LIN {X 0,Y 491.423,Z 544.675,A -85,B 0,C 180,E1 -6389.515,E2 -6389.515} C_VEL
LIN {X 0,Y 491.33,Z 557.602,A -85,B 0,C 180,E1 -6389.873,E2 -6389.873} C_VEL
LIN {X 0,Y 491.207,Z 570.582,A -85,B 0,C 180,E1 -6390.411,E2 -6390.411} C_VEL
LIN {X 0,Y 490.93,Z 581.621,A -85,B 0,C 180,E1 -6391.027,E2 -6391.027} C_VEL
LIN {X 0,Y 490.598,Z 593.027,A -85,B 0,C 180,E1 -6391.848,E2 -6391.848} C_VEL
LIN {X 0,Y 490.2,Z 603.319,A -85,B 0,C 180,E1 -6392.775,E2 -6392.775} C_VEL
LIN {X 0,Y 489.929,Z 611.716,A -85,B 0,C 180,E1 -6393.702,E2 -6393.702} C_VEL
LIN {X 0,Y 489.605,Z 619.489,A -85,B 0,C 180,E1 -6394.736,E2 -6394.736} C_VEL
LIN {X 0,Y 489.353,Z 627.085,A -85,B 0,C 180,E1 -6395.978,E2 -6395.978} C_VEL
LIN {X 0,Y 489.038,Z 634.088,A -85,B 0,C 180,E1 -6397.433,E2 -6397.433} C_VEL
LIN {X 0,Y 488.829,Z 638.765,A -85,B 0,C 180,E1 -6398.684,E2 -6398.684} C_VEL
LIN {X 0,Y 488.661,Z 642.349,A -85,B 0,C 180,E1 -6399.94,E2 -6399.94} C_VEL
LIN {X 0,Y 488.576,Z 644.196,A -85,B 0,C 180,E1 -6400.779,E2 -6400.779} C_VEL
LIN {X 0,Y 488.544,Z 646.052,A -85,B 0,C 180,E1 -6401.981,E2 -6401.981} C_VEL
LIN {X 0,Y 488.468,Z 647.149,A -85,B 0,C 180,E1 -6403.31,E2 -6403.31} C_VEL
LIN {X 0,Y 488.452,Z 647.319,A -85,B 0,C 180,E1 -6404.16,E2 -6404.16} C_VEL
LIN {X 0,Y 488.511,Z 646.803,A -85,B 0,C 180,E1 -6405.443,E2 -6405.443} C_VEL
LIN {X 0,Y 488.57,Z 645.357,A -85,B 0,C 180,E1 -6406.721,E2 -6406.721} C_VEL
LIN {X 0,Y 488.722,Z 642.05,A -85,B 0,C 180,E1 -6408.36,E2 -6408.36} C_VEL
LIN {X 0,Y 488.93,Z 637.94,A -85,B 0,C 180,E1 -6409.744,E2 -6409.744} C_VEL
LIN {X 0,Y 489.167,Z 632.802,A -85,B 0,C 180,E1 -6411.051,E2 -6411.051} C_VEL
LIN {X 0,Y 489.426,Z 626.172,A -85,B 0,C 180,E1 -6412.368,E2 -6412.368} C_VEL
LIN {X 0,Y 489.828,Z 617.767,A -85,B 0,C 180,E1 -6413.688,E2 -6413.688} C_VEL
LIN {X 0,Y 490.199,Z 609.017,A -85,B 0,C 180,E1 -6414.795,E2 -6414.795} C_VEL
LIN {X 0,Y 490.541,Z 599.188,A -85,B 0,C 180,E1 -6415.798,E2 -6415.798} C_VEL
LIN {X 0,Y 490.907,Z 588.286,A -85,B 0,C 180,E1 -6416.692,E2 -6416.692} C_VEL
LIN {X 0,Y 491.228,Z 577.789,A -85,B 0,C 180,E1 -6417.376,E2 -6417.376} C_VEL
LIN {X 0,Y 491.424,Z 565.398,A -85,B 0,C 180,E1 -6417.997,E2 -6417.997} C_VEL
LIN {X 0,Y 491.551,Z 552.8,A -85,B 0,C 180,E1 -6418.445,E2 -6418.445} C_VEL
LIN {X 0,Y 491.61,Z 539.967,A -85,B 0,C 180,E1 -6418.732,E2 -6418.732} C_VEL
LIN {X 0,Y 491.994,Z 472.881,A -85,B 0,C 180,E1 -6419.731,E2 -6419.731} C_VEL
LIN {X 0,Y 488.922,Z 464.493,A -85,B 0,C 180,E1 -6420.005,E2 -6420.005} C_VEL
LIN {X 0,Y 488.757,Z 463.677,A -85,B 0,C 180,E1 -6420.17,E2 -6420.17} C_VEL
LIN {X 0,Y 488.732,Z 463.606,A -85,B 0,C 180,E1 -6423.484,E2 -6423.484} C_VEL
LIN {X 0,Y 488.685,Z 463.613,A -85,B 0,C 180,E1 -6426.355,E2 -6426.355} C_VEL
LIN {X 0,Y 488.704,Z 463.606,A -85,B 0,C 180,E1 -6429.255,E2 -6429.255} C_VEL
LIN {X 0,Y 488.711,Z 463.605,A -85,B 0,C 180,E1 -6431.601,E2 -6431.601} C_VEL
LIN {X 0,Y 488.706,Z 463.613,A -85,B 0,C 180,E1 -6434.804,E2 -6434.804} C_VEL
LIN {X 0,Y 488.696,Z 463.61,A -85,B 0,C 180,E1 -6437.475,E2 -6437.475} C_VEL
LIN {X 0,Y 488.738,Z 463.606,A -85,B 0,C 180,E1 -6439.677,E2 -6439.677} C_VEL
LIN {X 0,Y 488.775,Z 463.798,A -85,B 0,C 180,E1 -6442.058,E2 -6442.058} C_VEL
LIN {X 0,Y 490.787,Z 474.144,A -85,B 0,C 180,E1 -6443.831,E2 -6443.831} C_VEL
LIN {X 0,Y 490.488,Z 489.742,A -85,B 0,C 180,E1 -6446.311,E2 -6446.311} C_VEL
LIN {X 0,Y 489.94,Z 509.149,A -85,B 0,C 180,E1 -6449.394,E2 -6449.394} C_VEL
LIN {X 0,Y 489.799,Z 518.237,A -85,B 0,C 180,E1 -6450.801,E2 -6450.801} C_VEL
LIN {X 0,Y 491.769,Z 530.283,A -85,B 0,C 180,E1 -6451.078,E2 -6451.078} C_VEL
LIN {X 0,Y 491.009,Z 626.779,A -85,B 0,C 180,E1 -6452.579,E2 -6452.579} C_VEL
LIN {X 0,Y 490.736,Z 640.314,A -85,B 0,C 180,E1 -6452.955,E2 -6452.955} C_VEL
LIN {X 0,Y 490.385,Z 653.402,A -85,B 0,C 180,E1 -6453.509,E2 -6453.509} C_VEL
LIN {X 0,Y 490.075,Z 665.153,A -85,B 0,C 180,E1 -6454.177,E2 -6454.177} C_VEL
LIN {X 0,Y 489.69,Z 676.455,A -85,B 0,C 180,E1 -6455.007,E2 -6455.007} C_VEL
LIN {X 0,Y 489.259,Z 686.707,A -85,B 0,C 180,E1 -6455.947,E2 -6455.947} C_VEL
LIN {X 0,Y 488.963,Z 695.329,A -85,B 0,C 180,E1 -6456.912,E2 -6456.912} C_VEL
LIN {X 0,Y 488.674,Z 703.624,A -85,B 0,C 180,E1 -6458.042,E2 -6458.042} C_VEL
LIN {X 0,Y 488.354,Z 711.06,A -85,B 0,C 180,E1 -6459.3,E2 -6459.3} C_VEL
LIN {X 0,Y 488.216,Z 717.473,A -85,B 0,C 180,E1 -6460.665,E2 -6460.665} C_VEL
LIN {X 0,Y 488.079,Z 721.901,A -85,B 0,C 180,E1 -6461.873,E2 -6461.873} C_VEL
LIN {X 0,Y 487.931,Z 725.713,A -85,B 0,C 180,E1 -6463.258,E2 -6463.258} C_VEL
LIN {X 0,Y 487.881,Z 728.525,A -85,B 0,C 180,E1 -6464.832,E2 -6464.832} C_VEL
LIN {X 0,Y 487.862,Z 729.56,A -85,B 0,C 180,E1 -6465.825,E2 -6465.825} C_VEL
LIN {X 0,Y 487.853,Z 729.953,A -85,B 0,C 180,E1 -6466.674,E2 -6466.674} C_VEL
LIN {X 0,Y 487.866,Z 729.946,A -85,B 0,C 180,E1 -6467.521,E2 -6467.521} C_VEL
LIN {X 0,Y 487.954,Z 729.524,A -85,B 0,C 180,E1 -6468.367,E2 -6468.367} C_VEL
LIN {X 0,Y 487.944,Z 728.654,A -85,B 0,C 180,E1 -6469.208,E2 -6469.208} C_VEL
LIN {X 0,Y 487.925,Z 727.388,A -85,B 0,C 180,E1 -6470.047,E2 -6470.047} C_VEL
LIN {X 0,Y 488.016,Z 724.667,A -85,B 0,C 180,E1 -6471.303,E2 -6471.303} C_VEL
LIN {X 0,Y 488.143,Z 720.913,A -85,B 0,C 180,E1 -6472.555,E2 -6472.555} C_VEL
LIN {X 0,Y 488.281,Z 715.569,A -85,B 0,C 180,E1 -6473.911,E2 -6473.911} C_VEL
LIN {X 0,Y 488.438,Z 708.705,A -85,B 0,C 180,E1 -6475.255,E2 -6475.255} C_VEL
LIN {X 0,Y 488.753,Z 700.753,A -85,B 0,C 180,E1 -6476.497,E2 -6476.497} C_VEL
LIN {X 0,Y 489.085,Z 692.626,A -85,B 0,C 180,E1 -6477.53,E2 -6477.53} C_VEL
LIN {X 0,Y 489.444,Z 682.634,A -85,B 0,C 180,E1 -6478.56,E2 -6478.56} C_VEL
LIN {X 0,Y 489.851,Z 671.472,A -85,B 0,C 180,E1 -6479.487,E2 -6479.487} C_VEL
LIN {X 0,Y 490.217,Z 660.49,A -85,B 0,C 180,E1 -6480.206,E2 -6480.206} C_VEL
LIN {X 0,Y 490.542,Z 648.224,A -85,B 0,C 180,E1 -6480.821,E2 -6480.821} C_VEL
LIN {X 0,Y 490.786,Z 635.579,A -85,B 0,C 180,E1 -6481.282,E2 -6481.282} C_VEL
LIN {X 0,Y 490.993,Z 621.991,A -85,B 0,C 180,E1 -6481.589,E2 -6481.589} C_VEL
LIN {X 0,Y 491.668,Z 529.585,A -85,B 0,C 180,E1 -6483.035,E2 -6483.035} C_VEL
LIN {X 0,Y 489.964,Z 519.063,A -85,B 0,C 180,E1 -6483.289,E2 -6483.289} C_VEL
LIN {X 0,Y 490.304,Z 499.165,A -85,B 0,C 180,E1 -6486.378,E2 -6486.378} C_VEL
LIN {X 0,Y 490.632,Z 482.876,A -85,B 0,C 180,E1 -6488.888,E2 -6488.888} C_VEL
LIN {X 0,Y 490.643,Z 473.536,A -85,B 0,C 180,E1 -6490.315,E2 -6490.315} C_VEL
LIN {X 0,Y 488.833,Z 463.701,A -85,B 0,C 180,E1 -6491.932,E2 -6491.932} C_VEL
LIN {X 0,Y 488.784,Z 463.602,A -85,B 0,C 180,E1 -6495.554,E2 -6495.554} C_VEL
LIN {X 0,Y 488.754,Z 463.604,A -85,B 0,C 180,E1 -6498.442,E2 -6498.442} C_VEL
LIN {X 0,Y 488.715,Z 463.612,A -85,B 0,C 180,E1 -6501.071,E2 -6501.071} C_VEL
LIN {X 0,Y 488.679,Z 463.611,A -85,B 0,C 180,E1 -6503.746,E2 -6503.746} C_VEL
LIN {X 0,Y 488.756,Z 463.606,A -85,B 0,C 180,E1 -6506.933,E2 -6506.933} C_VEL
LIN {X 0,Y 488.731,Z 463.606,A -85,B 0,C 180,E1 -6509.27,E2 -6509.27} C_VEL
LIN {X 0,Y 488.711,Z 463.607,A -85,B 0,C 180,E1 -6512.147,E2 -6512.147} C_VEL
LIN {X 0,Y 488.726,Z 463.606,A -85,B 0,C 180,E1 -6515.115,E2 -6515.115} C_VEL
LIN {X 0,Y 488.688,Z 463.612,A -85,B 0,C 180,E1 -6518.2,E2 -6518.2} C_VEL
LIN {X 0,Y 488.727,Z 463.608,A -85,B 0,C 180,E1 -6520.344,E2 -6520.344} C_VEL
LIN {X 0,Y 488.692,Z 463.609,A -85,B 0,C 180,E1 -6523.654,E2 -6523.654} C_VEL
LIN {X 0,Y 488.692,Z 463.613,A -85,B 0,C 180,E1 -6526.345,E2 -6526.345} C_VEL
LIN {X 0,Y 488.741,Z 463.604,A -85,B 0,C 180,E1 -6529.676,E2 -6529.676} C_VEL
LIN {X 0,Y 488.677,Z 463.61,A -85,B 0,C 180,E1 -6532.84,E2 -6532.84} C_VEL
LIN {X 0,Y 488.725,Z 463.599,A -85,B 0,C 180,E1 -6535.885,E2 -6535.885} C_VEL
LIN {X 0,Y 488.698,Z 463.611,A -85,B 0,C 180,E1 -6538.819,E2 -6538.819} C_VEL
LIN {X 0,Y 488.799,Z 463.817,A -85,B 0,C 180,E1 -6540.334,E2 -6540.334} C_VEL
LIN {X 0,Y 492.029,Z 478.714,A -85,B 0,C 180,E1 -6542.534,E2 -6542.534} C_VEL
LIN {X 0,Y 491.86,Z 487.643,A -85,B 0,C 180,E1 -6543.707,E2 -6543.707} C_VEL
LIN {X 0,Y 491.059,Z 510.131,A -85,B 0,C 180,E1 -6546.598,E2 -6546.598} C_VEL
LIN {X 0,Y 490.338,Z 532.663,A -85,B 0,C 180,E1 -6549.441,E2 -6549.441} C_VEL
LIN {X 0,Y 489.667,Z 556.938,A -85,B 0,C 180,E1 -6552.457,E2 -6552.457} C_VEL
LIN {X 0,Y 489.448,Z 567.191,A -85,B 0,C 180,E1 -6553.696,E2 -6553.696} C_VEL
LIN {X 0,Y 491.565,Z 587.846,A -85,B 0,C 180,E1 -6554.086,E2 -6554.086} C_VEL
LIN {X 0,Y 491.001,Z 678.547,A -85,B 0,C 180,E1 -6555.439,E2 -6555.439} C_VEL
LIN {X 0,Y 490.587,Z 692.383,A -85,B 0,C 180,E1 -6555.824,E2 -6555.824} C_VEL
LIN {X 0,Y 490.217,Z 705.371,A -85,B 0,C 180,E1 -6556.368,E2 -6556.368} C_VEL
LIN {X 0,Y 489.788,Z 717.734,A -85,B 0,C 180,E1 -6557.074,E2 -6557.074} C_VEL
LIN {X 0,Y 489.444,Z 728.753,A -85,B 0,C 180,E1 -6557.876,E2 -6557.876} C_VEL
LIN {X 0,Y 488.951,Z 739.13,A -85,B 0,C 180,E1 -6558.81,E2 -6558.81} C_VEL
LIN {X 0,Y 488.72,Z 748.521,A -85,B 0,C 180,E1 -6559.853,E2 -6559.853} C_VEL
LIN {X 0,Y 488.44,Z 757.666,A -85,B 0,C 180,E1 -6561.101,E2 -6561.101} C_VEL
LIN {X 0,Y 488.243,Z 765.039,A -85,B 0,C 180,E1 -6562.347,E2 -6562.347} C_VEL
LIN {X 0,Y 488.133,Z 771.508,A -85,B 0,C 180,E1 -6563.686,E2 -6563.686} C_VEL
LIN {X 0,Y 488.082,Z 776.557,A -85,B 0,C 180,E1 -6565.042,E2 -6565.042} C_VEL
LIN {X 0,Y 488.135,Z 778.96,A -85,B 0,C 180,E1 -6565.87,E2 -6565.87} C_VEL
LIN {X 0,Y 488.074,Z 780.886,A -85,B 0,C 180,E1 -6566.697,E2 -6566.697} C_VEL
LIN {X 0,Y 488.067,Z 782.375,A -85,B 0,C 180,E1 -6567.523,E2 -6567.523} C_VEL
LIN {X 0,Y 488.009,Z 783.436,A -85,B 0,C 180,E1 -6568.348,E2 -6568.348} C_VEL
LIN {X 0,Y 487.983,Z 784.079,A -85,B 0,C 180,E1 -6569.173,E2 -6569.173} C_VEL
LIN {X 0,Y 488.043,Z 784.312,A -85,B 0,C 180,E1 -6569.999,E2 -6569.999} C_VEL
LIN {X 0,Y 487.98,Z 784.11,A -85,B 0,C 180,E1 -6570.824,E2 -6570.824} C_VEL
LIN {X 0,Y 488.003,Z 783.495,A -85,B 0,C 180,E1 -6571.649,E2 -6571.649} C_VEL
LIN {X 0,Y 488.061,Z 782.466,A -85,B 0,C 180,E1 -6572.475,E2 -6572.475} C_VEL
LIN {X 0,Y 488.067,Z 781.001,A -85,B 0,C 180,E1 -6573.301,E2 -6573.301} C_VEL
LIN {X 0,Y 488.05,Z 777.918,A -85,B 0,C 180,E1 -6574.541,E2 -6574.541} C_VEL
LIN {X 0,Y 488.18,Z 772.758,A -85,B 0,C 180,E1 -6576.046,E2 -6576.046} C_VEL
LIN {X 0,Y 488.205,Z 766.364,A -85,B 0,C 180,E1 -6577.443,E2 -6577.443} C_VEL
LIN {X 0,Y 488.389,Z 759.172,A -85,B 0,C 180,E1 -6578.689,E2 -6578.689} C_VEL
LIN {X 0,Y 488.632,Z 750.351,A -85,B 0,C 180,E1 -6579.937,E2 -6579.937} C_VEL
LIN {X 0,Y 488.956,Z 741.346,A -85,B 0,C 180,E1 -6580.977,E2 -6580.977} C_VEL
LIN {X 0,Y 489.354,Z 731.482,A -85,B 0,C 180,E1 -6581.913,E2 -6581.913} C_VEL
LIN {X 0,Y 489.709,Z 720.852,A -85,B 0,C 180,E1 -6582.735,E2 -6582.735} C_VEL
LIN {X 0,Y 490.113,Z 708.68,A -85,B 0,C 180,E1 -6583.473,E2 -6583.473} C_VEL
LIN {X 0,Y 490.512,Z 696.213,A -85,B 0,C 180,E1 -6584.043,E2 -6584.043} C_VEL
LIN {X 0,Y 490.892,Z 683.439,A -85,B 0,C 180,E1 -6584.455,E2 -6584.455} C_VEL
LIN {X 0,Y 491.073,Z 670.047,A -85,B 0,C 180,E1 -6584.715,E2 -6584.715} C_VEL
LIN {X 0,Y 491.533,Z 585.726,A -85,B 0,C 180,E1 -6585.951,E2 -6585.951} C_VEL
LIN {X 0,Y 489.464,Z 567.613,A -85,B 0,C 180,E1 -6586.301,E2 -6586.301} C_VEL
LIN {X 0,Y 489.986,Z 545.924,A -85,B 0,C 180,E1 -6588.965,E2 -6588.965} C_VEL
LIN {X 0,Y 490.885,Z 517.599,A -85,B 0,C 180,E1 -6592.517,E2 -6592.517} C_VEL
LIN {X 0,Y 491.631,Z 493.909,A -85,B 0,C 180,E1 -6595.531,E2 -6595.531} C_VEL
LIN {X 0,Y 492.066,Z 478.853,A -85,B 0,C 180,E1 -6597.477,E2 -6597.477} C_VEL
LIN {X 0,Y 488.75,Z 463.732,A -85,B 0,C 180,E1 -6599.666,E2 -6599.666} C_VEL
LIN {X 0,Y 488.73,Z 463.606,A -85,B 0,C 180,E1 -6603.121,E2 -6603.121} C_VEL
LIN {X 0,Y 488.658,Z 463.619,A -85,B 0,C 180,E1 -6606.132,E2 -6606.132} C_VEL
LIN {X 0,Y 488.68,Z 463.608,A -85,B 0,C 180,E1 -6609.254,E2 -6609.254} C_VEL
LIN {X 0,Y 488.658,Z 463.615,A -85,B 0,C 180,E1 -6612.527,E2 -6612.527} C_VEL
LIN {X 0,Y 488.692,Z 463.606,A -85,B 0,C 180,E1 -6615.196,E2 -6615.196} C_VEL
LIN {X 0,Y 488.67,Z 463.613,A -85,B 0,C 180,E1 -6618.58,E2 -6618.58} C_VEL
LIN {X 0,Y 488.664,Z 463.612,A -85,B 0,C 180,E1 -6621.798,E2 -6621.798} C_VEL
LIN {X 0,Y 488.711,Z 463.604,A -85,B 0,C 180,E1 -6625.051,E2 -6625.051} C_VEL
LIN {X 0,Y 488.692,Z 463.611,A -85,B 0,C 180,E1 -6628.045,E2 -6628.045} C_VEL
LIN {X 0,Y 488.71,Z 463.607,A -85,B 0,C 180,E1 -6630.728,E2 -6630.728} C_VEL
LIN {X 0,Y 488.723,Z 463.603,A -85,B 0,C 180,E1 -6633.526,E2 -6633.526} C_VEL
LIN {X 0,Y 488.659,Z 463.617,A -85,B 0,C 180,E1 -6636.252,E2 -6636.252} C_VEL
LIN {X 0,Y 488.733,Z 463.601,A -85,B 0,C 180,E1 -6639.175,E2 -6639.175} C_VEL
LIN {X 0,Y 488.714,Z 463.613,A -85,B 0,C 180,E1 -6642.422,E2 -6642.422} C_VEL
LIN {X 0,Y 488.747,Z 463.601,A -85,B 0,C 180,E1 -6644.999,E2 -6644.999} C_VEL
LIN {X 0,Y 488.795,Z 463.601,A -85,B 0,C 180,E1 -6648.387,E2 -6648.387} C_VEL
LIN {X 0,Y 488.802,Z 463.593,A -85,B 0,C 180,E1 -6651.733,E2 -6651.733} C_VEL
LIN {X 0,Y 488.829,Z 463.594,A -85,B 0,C 180,E1 -6654.224,E2 -6654.224} C_VEL
LIN {X 0,Y 488.945,Z 463.575,A -85,B 0,C 180,E1 -6657.528,E2 -6657.528} C_VEL
LIN {X 0,Y 488.962,Z 463.577,A -85,B 0,C 180,E1 -6660.823,E2 -6660.823} C_VEL
LIN {X 0,Y 488.946,Z 463.582,A -85,B 0,C 180,E1 -6662.471,E2 -6662.471} C_VEL
LIN {X 0,Y 488.833,Z 463.589,A -85,B 0,C 180,E1 -6665.776,E2 -6665.776} C_VEL
LIN {X 0,Y 488.804,Z 463.596,A -85,B 0,C 180,E1 -6668.266,E2 -6668.266} C_VEL
LIN {X 0,Y 488.794,Z 463.593,A -85,B 0,C 180,E1 -6671.612,E2 -6671.612} C_VEL
LIN {X 0,Y 488.75,Z 463.603,A -85,B 0,C 180,E1 -6675,E2 -6675} C_VEL
LIN {X 0,Y 488.74,Z 463.605,A -85,B 0,C 180,E1 -6678.442,E2 -6678.442} C_VEL
LIN {X 0,Y 488.694,Z 463.61,A -85,B 0,C 180,E1 -6681.071,E2 -6681.071} C_VEL
LIN {X 0,Y 488.679,Z 463.608,A -85,B 0,C 180,E1 -6683.746,E2 -6683.746} C_VEL
LIN {X 0,Y 488.785,Z 463.601,A -85,B 0,C 180,E1 -6686.946,E2 -6686.946} C_VEL
LIN {X 0,Y 488.696,Z 463.609,A -85,B 0,C 180,E1 -6690.364,E2 -6690.364} C_VEL
LIN {X 0,Y 488.723,Z 463.603,A -85,B 0,C 180,E1 -6693.485,E2 -6693.485} C_VEL
LIN {X 0,Y 488.676,Z 463.611,A -85,B 0,C 180,E1 -6696.356,E2 -6696.356} C_VEL
LIN {X 0,Y 488.689,Z 463.61,A -85,B 0,C 180,E1 -6699.255,E2 -6699.255} C_VEL
LIN {X 0,Y 488.711,Z 463.604,A -85,B 0,C 180,E1 -6701.603,E2 -6701.603} C_VEL
LIN {X 0,Y 488.7,Z 463.613,A -85,B 0,C 180,E1 -6704.802,E2 -6704.802} C_VEL
LIN {X 0,Y 488.723,Z 463.604,A -85,B 0,C 180,E1 -6707.48,E2 -6707.48} C_VEL
LIN {X 0,Y 488.739,Z 463.607,A -85,B 0,C 180,E1 -6710.752,E2 -6710.752} C_VEL
LIN {X 0,Y 488.674,Z 463.608,A -85,B 0,C 180,E1 -6713.87,E2 -6713.87} C_VEL
LIN {X 0,Y 488.731,Z 463.609,A -85,B 0,C 180,E1 -6716.879,E2 -6716.879} C_VEL
LIN {X 0,Y 488.716,Z 463.603,A -85,B 0,C 180,E1 -6719.782,E2 -6719.782} C_VEL
LIN {X 0,Y 488.785,Z 463.603,A -85,B 0,C 180,E1 -6723.058,E2 -6723.058} C_VEL
LIN {X 0,Y 488.736,Z 463.602,A -85,B 0,C 180,E1 -6724.363,E2 -6724.363} C_VEL
LIN {X 0,Y 488.093,Z 463.69,A -85,B 0,C 180,E1 -6725.051,E2 -6725.051} C_VEL
LIN {X 0,Y 485.223,Z 464.043,A -85,B 0,C 180,E1 -6726.168,E2 -6726.168} C_VEL
LIN {X 0,Y 482.776,Z 464.352,A -85,B 0,C 180,E1 -6727.068,E2 -6727.068} C_VEL
LIN {X 0,Y 481.718,Z 464.476,A -85,B 0,C 180,E1 -6727.763,E2 -6727.763} C_VEL
LIN {X 0,Y 481.63,Z 464.486,A -85,B 0,C 180,E1 -6727.999,E2 -6727.999} C_VEL
LIN {X 0,Y 481.702,Z 464.478,A -85,B 0,C 180,E1 -6730.395,E2 -6730.395} C_VEL
LIN {X 0,Y 481.687,Z 464.487,A -85,B 0,C 180,E1 -6733.035,E2 -6733.035} C_VEL
LIN {X 0,Y 481.686,Z 464.481,A -85,B 0,C 180,E1 -6735.64,E2 -6735.64} C_VEL
LIN {X 0,Y 481.747,Z 464.471,A -85,B 0,C 180,E1 -6738.217,E2 -6738.217} C_VEL
LIN {X 0,Y 481.76,Z 464.475,A -85,B 0,C 180,E1 -6741.613,E2 -6741.613} C_VEL
LIN {X 0,Y 481.817,Z 464.467,A -85,B 0,C 180,E1 -6744.141,E2 -6744.141} C_VEL
LIN {X 0,Y 481.885,Z 464.583,A -85,B 0,C 180,E1 -6747.839,E2 -6747.839} C_VEL
LIN {X 0,Y 482.07,Z 465.64,A -85,B 0,C 180,E1 -6747.996,E2 -6747.996} C_VEL
LIN {X 0,Y 484.988,Z 474.293,A -85,B 0,C 180,E1 -6748.235,E2 -6748.235} C_VEL
LIN {X 0,Y 484.58,Z 545.83,A -85,B 0,C 180,E1 -6749.326,E2 -6749.326} C_VEL
LIN {X 0,Y 484.488,Z 558.693,A -85,B 0,C 180,E1 -6749.69,E2 -6749.69} C_VEL
LIN {X 0,Y 484.358,Z 571.103,A -85,B 0,C 180,E1 -6750.209,E2 -6750.209} C_VEL
LIN {X 0,Y 484.066,Z 582.267,A -85,B 0,C 180,E1 -6750.833,E2 -6750.833} C_VEL
LIN {X 0,Y 483.712,Z 593.755,A -85,B 0,C 180,E1 -6751.667,E2 -6751.667} C_VEL
LIN {X 0,Y 483.302,Z 604.094,A -85,B 0,C 180,E1 -6752.606,E2 -6752.606} C_VEL
LIN {X 0,Y 483.018,Z 612.523,A -85,B 0,C 180,E1 -6753.547,E2 -6753.547} C_VEL
LIN {X 0,Y 482.672,Z 620.324,A -85,B 0,C 180,E1 -6754.595,E2 -6754.595} C_VEL
LIN {X 0,Y 482.376,Z 627.962,A -85,B 0,C 180,E1 -6755.855,E2 -6755.855} C_VEL
LIN {X 0,Y 482.083,Z 634.595,A -85,B 0,C 180,E1 -6757.239,E2 -6757.239} C_VEL
LIN {X 0,Y 481.806,Z 640.371,A -85,B 0,C 180,E1 -6758.812,E2 -6758.812} C_VEL
LIN {X 0,Y 481.634,Z 643.8,A -85,B 0,C 180,E1 -6760.086,E2 -6760.086} C_VEL
LIN {X 0,Y 481.538,Z 645.51,A -85,B 0,C 180,E1 -6760.939,E2 -6760.939} C_VEL
LIN {X 0,Y 481.522,Z 647.165,A -85,B 0,C 180,E1 -6762.072,E2 -6762.072} C_VEL
LIN {X 0,Y 481.455,Z 648.2,A -85,B 0,C 180,E1 -6763.508,E2 -6763.508} C_VEL
LIN {X 0,Y 481.426,Z 648.271,A -85,B 0,C 180,E1 -6764.371,E2 -6764.371} C_VEL
LIN {X 0,Y 481.496,Z 647.711,A -85,B 0,C 180,E1 -6765.562,E2 -6765.562} C_VEL
LIN {X 0,Y 481.58,Z 646.015,A -85,B 0,C 180,E1 -6766.971,E2 -6766.971} C_VEL
LIN {X 0,Y 481.738,Z 642.857,A -85,B 0,C 180,E1 -6768.51,E2 -6768.51} C_VEL
LIN {X 0,Y 481.99,Z 638.244,A -85,B 0,C 180,E1 -6770.04,E2 -6770.04} C_VEL
LIN {X 0,Y 482.244,Z 632.868,A -85,B 0,C 180,E1 -6771.368,E2 -6771.368} C_VEL
LIN {X 0,Y 482.591,Z 626.011,A -85,B 0,C 180,E1 -6772.702,E2 -6772.702} C_VEL
LIN {X 0,Y 482.943,Z 618.522,A -85,B 0,C 180,E1 -6773.876,E2 -6773.876} C_VEL
LIN {X 0,Y 483.322,Z 610.208,A -85,B 0,C 180,E1 -6774.943,E2 -6774.943} C_VEL
LIN {X 0,Y 483.687,Z 600.444,A -85,B 0,C 180,E1 -6775.96,E2 -6775.96} C_VEL
LIN {X 0,Y 484.085,Z 589.615,A -85,B 0,C 180,E1 -6776.865,E2 -6776.865} C_VEL
LIN {X 0,Y 484.411,Z 579.41,A -85,B 0,C 180,E1 -6777.547,E2 -6777.547} C_VEL
LIN {X 0,Y 484.645,Z 568.151,A -85,B 0,C 180,E1 -6778.137,E2 -6778.137} C_VEL
LIN {X 0,Y 484.766,Z 555.689,A -85,B 0,C 180,E1 -6778.613,E2 -6778.613} C_VEL
LIN {X 0,Y 484.823,Z 542.482,A -85,B 0,C 180,E1 -6778.934,E2 -6778.934} C_VEL
LIN {X 0,Y 485.23,Z 474.35,A -85,B 0,C 180,E1 -6779.969,E2 -6779.969} C_VEL
LIN {X 0,Y 481.901,Z 465.577,A -85,B 0,C 180,E1 -6780.255,E2 -6780.255} C_VEL
LIN {X 0,Y 481.681,Z 464.581,A -85,B 0,C 180,E1 -6780.424,E2 -6780.424} C_VEL
LIN {X 0,Y 481.678,Z 464.484,A -85,B 0,C 180,E1 -6783.73,E2 -6783.73} C_VEL
LIN {X 0,Y 481.629,Z 464.492,A -85,B 0,C 180,E1 -6786.748,E2 -6786.748} C_VEL
LIN {X 0,Y 481.681,Z 464.479,A -85,B 0,C 180,E1 -6789.941,E2 -6789.941} C_VEL
LIN {X 0,Y 481.636,Z 464.491,A -85,B 0,C 180,E1 -6793.148,E2 -6793.148} C_VEL
LIN {X 0,Y 481.658,Z 464.485,A -85,B 0,C 180,E1 -6795.642,E2 -6795.642} C_VEL
LIN {X 0,Y 481.661,Z 464.491,A -85,B 0,C 180,E1 -6798.959,E2 -6798.959} C_VEL
LIN {X 0,Y 481.738,Z 464.702,A -85,B 0,C 180,E1 -6801.864,E2 -6801.864} C_VEL
LIN {X 0,Y 483.873,Z 475.473,A -85,B 0,C 180,E1 -6803.711,E2 -6803.711} C_VEL
LIN {X 0,Y 483.569,Z 491.007,A -85,B 0,C 180,E1 -6806.203,E2 -6806.203} C_VEL
LIN {X 0,Y 483.022,Z 509.39,A -85,B 0,C 180,E1 -6809.145,E2 -6809.145} C_VEL
LIN {X 0,Y 482.83,Z 518.311,A -85,B 0,C 180,E1 -6810.546,E2 -6810.546} C_VEL
LIN {X 0,Y 484.098,Z 525.738,A -85,B 0,C 180,E1 -6810.743,E2 -6810.743} C_VEL
LIN {X 0,Y 484.911,Z 531.562,A -85,B 0,C 180,E1 -6810.865,E2 -6810.865} C_VEL
LIN {X 0,Y 484.112,Z 626.805,A -85,B 0,C 180,E1 -6812.378,E2 -6812.378} C_VEL
LIN {X 0,Y 483.834,Z 639.961,A -85,B 0,C 180,E1 -6812.741,E2 -6812.741} C_VEL
LIN {X 0,Y 483.48,Z 652.693,A -85,B 0,C 180,E1 -6813.275,E2 -6813.275} C_VEL
LIN {X 0,Y 483.139,Z 665.57,A -85,B 0,C 180,E1 -6814.01,E2 -6814.01} C_VEL
LIN {X 0,Y 482.72,Z 677.046,A -85,B 0,C 180,E1 -6814.868,E2 -6814.868} C_VEL
LIN {X 0,Y 482.271,Z 687.112,A -85,B 0,C 180,E1 -6815.804,E2 -6815.804} C_VEL
LIN {X 0,Y 481.955,Z 695.982,A -85,B 0,C 180,E1 -6816.814,E2 -6816.814} C_VEL
LIN {X 0,Y 481.655,Z 704.031,A -85,B 0,C 180,E1 -6817.931,E2 -6817.931} C_VEL
LIN {X 0,Y 481.342,Z 711.135,A -85,B 0,C 180,E1 -6819.143,E2 -6819.143} C_VEL
LIN {X 0,Y 481.171,Z 716.953,A -85,B 0,C 180,E1 -6820.371,E2 -6820.371} C_VEL
LIN {X 0,Y 481.017,Z 722.101,A -85,B 0,C 180,E1 -6821.752,E2 -6821.752} C_VEL
LIN {X 0,Y 480.875,Z 725.61,A -85,B 0,C 180,E1 -6823.005,E2 -6823.005} C_VEL
LIN {X 0,Y 480.83,Z 727.465,A -85,B 0,C 180,E1 -6823.877,E2 -6823.877} C_VEL
LIN {X 0,Y 480.796,Z 728.836,A -85,B 0,C 180,E1 -6824.745,E2 -6824.745} C_VEL
LIN {X 0,Y 480.795,Z 729.792,A -85,B 0,C 180,E1 -6825.612,E2 -6825.612} C_VEL
LIN {X 0,Y 480.76,Z 730.306,A -85,B 0,C 180,E1 -6826.474,E2 -6826.474} C_VEL
LIN {X 0,Y 480.779,Z 730.374,A -85,B 0,C 180,E1 -6827.334,E2 -6827.334} C_VEL
LIN {X 0,Y 480.859,Z 729.977,A -85,B 0,C 180,E1 -6828.309,E2 -6828.309} C_VEL
LIN {X 0,Y 480.859,Z 728.102,A -85,B 0,C 180,E1 -6829.899,E2 -6829.899} C_VEL
LIN {X 0,Y 480.941,Z 725.524,A -85,B 0,C 180,E1 -6831.174,E2 -6831.174} C_VEL
LIN {X 0,Y 481.067,Z 721.918,A -85,B 0,C 180,E1 -6832.445,E2 -6832.445} C_VEL
LIN {X 0,Y 481.224,Z 716.591,A -85,B 0,C 180,E1 -6833.856,E2 -6833.856} C_VEL
LIN {X 0,Y 481.383,Z 710.119,A -85,B 0,C 180,E1 -6835.185,E2 -6835.185} C_VEL
LIN {X 0,Y 481.681,Z 702.374,A -85,B 0,C 180,E1 -6836.445,E2 -6836.445} C_VEL
LIN {X 0,Y 482.039,Z 694.484,A -85,B 0,C 180,E1 -6837.493,E2 -6837.493} C_VEL
LIN {X 0,Y 482.397,Z 684.909,A -85,B 0,C 180,E1 -6838.539,E2 -6838.539} C_VEL
LIN {X 0,Y 482.808,Z 674.153,A -85,B 0,C 180,E1 -6839.479,E2 -6839.479} C_VEL
LIN {X 0,Y 483.255,Z 662.086,A -85,B 0,C 180,E1 -6840.313,E2 -6840.313} C_VEL
LIN {X 0,Y 483.63,Z 650.191,A -85,B 0,C 180,E1 -6840.937,E2 -6840.937} C_VEL
LIN {X 0,Y 483.907,Z 636.515,A -85,B 0,C 180,E1 -6841.457,E2 -6841.457} C_VEL
LIN {X 0,Y 484.092,Z 623.457,A -85,B 0,C 180,E1 -6841.768,E2 -6841.768} C_VEL
LIN {X 0,Y 484.876,Z 530.321,A -85,B 0,C 180,E1 -6843.259,E2 -6843.259} C_VEL
LIN {X 0,Y 483.077,Z 519.738,A -85,B 0,C 180,E1 -6843.519,E2 -6843.519} C_VEL
LIN {X 0,Y 483.07,Z 516.568,A -85,B 0,C 180,E1 -6843.963,E2 -6843.963} C_VEL
LIN {X 0,Y 483.58,Z 495.339,A -85,B 0,C 180,E1 -6847.306,E2 -6847.306} C_VEL
LIN {X 0,Y 483.894,Z 476.198,A -85,B 0,C 180,E1 -6850.249,E2 -6850.249} C_VEL
LIN {X 0,Y 481.801,Z 464.684,A -85,B 0,C 180,E1 -6852.123,E2 -6852.123} C_VEL
LIN {X 0,Y 481.732,Z 464.48,A -85,B 0,C 180,E1 -6855.658,E2 -6855.658} C_VEL
LIN {X 0,Y 481.715,Z 464.483,A -85,B 0,C 180,E1 -6858.722,E2 -6858.722} C_VEL
LIN {X 0,Y 481.653,Z 464.49,A -85,B 0,C 180,E1 -6861.395,E2 -6861.395} C_VEL
LIN {X 0,Y 481.658,Z 464.486,A -85,B 0,C 180,E1 -6864.114,E2 -6864.114} C_VEL
LIN {X 0,Y 481.724,Z 464.482,A -85,B 0,C 180,E1 -6867.132,E2 -6867.132} C_VEL
LIN {X 0,Y 481.686,Z 464.481,A -85,B 0,C 180,E1 -6869.741,E2 -6869.741} C_VEL
LIN {X 0,Y 481.68,Z 464.487,A -85,B 0,C 180,E1 -6872.674,E2 -6872.674} C_VEL
LIN {X 0,Y 481.645,Z 464.486,A -85,B 0,C 180,E1 -6875.709,E2 -6875.709} C_VEL
LIN {X 0,Y 481.679,Z 464.487,A -85,B 0,C 180,E1 -6878.859,E2 -6878.859} C_VEL
LIN {X 0,Y 481.66,Z 464.486,A -85,B 0,C 180,E1 -6881.912,E2 -6881.912} C_VEL
LIN {X 0,Y 481.663,Z 464.488,A -85,B 0,C 180,E1 -6884.457,E2 -6884.457} C_VEL
LIN {X 0,Y 481.655,Z 464.488,A -85,B 0,C 180,E1 -6887.839,E2 -6887.839} C_VEL
LIN {X 0,Y 481.666,Z 464.478,A -85,B 0,C 180,E1 -6890.654,E2 -6890.654} C_VEL
LIN {X 0,Y 481.629,Z 464.489,A -85,B 0,C 180,E1 -6893.377,E2 -6893.377} C_VEL
LIN {X 0,Y 481.677,Z 464.479,A -85,B 0,C 180,E1 -6896.326,E2 -6896.326} C_VEL
LIN {X 0,Y 481.741,Z 464.574,A -85,B 0,C 180,E1 -6900.021,E2 -6900.021} C_VEL
LIN {X 0,Y 482.364,Z 467.268,A -85,B 0,C 180,E1 -6900.488,E2 -6900.488} C_VEL
LIN {X 0,Y 485.125,Z 480,A -85,B 0,C 180,E1 -6902.38,E2 -6902.38} C_VEL
LIN {X 0,Y 485.108,Z 486.894,A -85,B 0,C 180,E1 -6903.312,E2 -6903.312} C_VEL
LIN {X 0,Y 484.106,Z 511.253,A -85,B 0,C 180,E1 -6906.497,E2 -6906.497} C_VEL
LIN {X 0,Y 483.276,Z 535.227,A -85,B 0,C 180,E1 -6909.571,E2 -6909.571} C_VEL
LIN {X 0,Y 482.573,Z 559.42,A -85,B 0,C 180,E1 -6912.628,E2 -6912.628} C_VEL
LIN {X 0,Y 482.419,Z 566.308,A -85,B 0,C 180,E1 -6913.451,E2 -6913.451} C_VEL
LIN {X 0,Y 484.718,Z 587.575,A -85,B 0,C 180,E1 -6913.864,E2 -6913.864} C_VEL
LIN {X 0,Y 484.117,Z 677.547,A -85,B 0,C 180,E1 -6915.228,E2 -6915.228} C_VEL
LIN {X 0,Y 483.647,Z 691.355,A -85,B 0,C 180,E1 -6915.616,E2 -6915.616} C_VEL
LIN {X 0,Y 483.276,Z 704.33,A -85,B 0,C 180,E1 -6916.169,E2 -6916.169} C_VEL
LIN {X 0,Y 482.849,Z 716.217,A -85,B 0,C 180,E1 -6916.853,E2 -6916.853} C_VEL
LIN {X 0,Y 482.476,Z 726.11,A -85,B 0,C 180,E1 -6917.568,E2 -6917.568} C_VEL
LIN {X 0,Y 481.972,Z 737.028,A -85,B 0,C 180,E1 -6918.539,E2 -6918.539} C_VEL
LIN {X 0,Y 481.719,Z 745.766,A -85,B 0,C 180,E1 -6919.491,E2 -6919.491} C_VEL
LIN {X 0,Y 481.379,Z 756.878,A -85,B 0,C 180,E1 -6920.969,E2 -6920.969} C_VEL
LIN {X 0,Y 481.169,Z 764.519,A -85,B 0,C 180,E1 -6922.234,E2 -6922.234} C_VEL
LIN {X 0,Y 481.035,Z 771.506,A -85,B 0,C 180,E1 -6923.704,E2 -6923.704} C_VEL
LIN {X 0,Y 481.007,Z 776.112,A -85,B 0,C 180,E1 -6924.969,E2 -6924.969} C_VEL
LIN {X 0,Y 481.027,Z 778.53,A -85,B 0,C 180,E1 -6925.809,E2 -6925.809} C_VEL
LIN {X 0,Y 480.999,Z 780.478,A -85,B 0,C 180,E1 -6926.648,E2 -6926.648} C_VEL
LIN {X 0,Y 481.001,Z 781.974,A -85,B 0,C 180,E1 -6927.486,E2 -6927.486} C_VEL
LIN {X 0,Y 480.934,Z 783.035,A -85,B 0,C 180,E1 -6928.324,E2 -6928.324} C_VEL
LIN {X 0,Y 480.9,Z 783.679,A -85,B 0,C 180,E1 -6929.161,E2 -6929.161} C_VEL
LIN {X 0,Y 480.954,Z 783.919,A -85,B 0,C 180,E1 -6929.999,E2 -6929.999} C_VEL
LIN {X 0,Y 480.897,Z 783.712,A -85,B 0,C 180,E1 -6930.836,E2 -6930.836} C_VEL
LIN {X 0,Y 480.929,Z 783.096,A -85,B 0,C 180,E1 -6931.673,E2 -6931.673} C_VEL
LIN {X 0,Y 480.995,Z 782.07,A -85,B 0,C 180,E1 -6932.511,E2 -6932.511} C_VEL
LIN {X 0,Y 480.991,Z 780.602,A -85,B 0,C 180,E1 -6933.349,E2 -6933.349} C_VEL
LIN {X 0,Y 480.959,Z 777.525,A -85,B 0,C 180,E1 -6934.608,E2 -6934.608} C_VEL
LIN {X 0,Y 481.061,Z 773.397,A -85,B 0,C 180,E1 -6935.868,E2 -6935.868} C_VEL
LIN {X 0,Y 481.114,Z 767.017,A -85,B 0,C 180,E1 -6937.342,E2 -6937.342} C_VEL
LIN {X 0,Y 481.304,Z 760.01,A -85,B 0,C 180,E1 -6938.606,E2 -6938.606} C_VEL
LIN {X 0,Y 481.52,Z 751.221,A -85,B 0,C 180,E1 -6939.873,E2 -6939.873} C_VEL
LIN {X 0,Y 481.939,Z 739.357,A -85,B 0,C 180,E1 -6941.246,E2 -6941.246} C_VEL
LIN {X 0,Y 482.381,Z 729.828,A -85,B 0,C 180,E1 -6942.147,E2 -6942.147} C_VEL
LIN {X 0,Y 482.697,Z 719.701,A -85,B 0,C 180,E1 -6942.934,E2 -6942.934} C_VEL
LIN {X 0,Y 483.141,Z 707.679,A -85,B 0,C 180,E1 -6943.671,E2 -6943.671} C_VEL
LIN {X 0,Y 483.589,Z 695.213,A -85,B 0,C 180,E1 -6944.248,E2 -6944.248} C_VEL
LIN {X 0,Y 484.004,Z 682.432,A -85,B 0,C 180,E1 -6944.665,E2 -6944.665} C_VEL
LIN {X 0,Y 484.21,Z 667.222,A -85,B 0,C 180,E1 -6944.955,E2 -6944.955} C_VEL
LIN {X 0,Y 484.706,Z 586.566,A -85,B 0,C 180,E1 -6946.153,E2 -6946.153} C_VEL
LIN {X 0,Y 482.425,Z 566.563,A -85,B 0,C 180,E1 -6946.546,E2 -6946.546} C_VEL
LIN {X 0,Y 483.103,Z 542.592,A -85,B 0,C 180,E1 -6949.546,E2 -6949.546} C_VEL
LIN {X 0,Y 483.903,Z 518.363,A -85,B 0,C 180,E1 -6952.634,E2 -6952.634} C_VEL
LIN {X 0,Y 484.663,Z 495.736,A -85,B 0,C 180,E1 -6955.555,E2 -6955.555} C_VEL
LIN {X 0,Y 485.266,Z 481.773,A -85,B 0,C 180,E1 -6957.374,E2 -6957.374} C_VEL
LIN {X 0,Y 483.909,Z 474.43,A -85,B 0,C 180,E1 -6958.412,E2 -6958.412} C_VEL
LIN {X 0,Y 481.708,Z 464.619,A -85,B 0,C 180,E1 -6959.873,E2 -6959.873} C_VEL
LIN {X 0,Y 481.665,Z 464.488,A -85,B 0,C 180,E1 -6962.673,E2 -6962.673} C_VEL
LIN {X 0,Y 481.622,Z 464.493,A -85,B 0,C 180,E1 -6965.709,E2 -6965.709} C_VEL
LIN {X 0,Y 481.624,Z 464.487,A -85,B 0,C 180,E1 -6968.861,E2 -6968.861} C_VEL
LIN {X 0,Y 481.626,Z 464.491,A -85,B 0,C 180,E1 -6971.909,E2 -6971.909} C_VEL
LIN {X 0,Y 481.645,Z 464.489,A -85,B 0,C 180,E1 -6974.457,E2 -6974.457} C_VEL
LIN {X 0,Y 481.631,Z 464.489,A -85,B 0,C 180,E1 -6977.837,E2 -6977.837} C_VEL
LIN {X 0,Y 481.655,Z 464.483,A -85,B 0,C 180,E1 -6981.139,E2 -6981.139} C_VEL
LIN {X 0,Y 481.649,Z 464.486,A -85,B 0,C 180,E1 -6984.795,E2 -6984.795} C_VEL
LIN {X 0,Y 481.66,Z 464.482,A -85,B 0,C 180,E1 -6987.325,E2 -6987.325} C_VEL
LIN {X 0,Y 481.666,Z 464.489,A -85,B 0,C 180,E1 -6990.258,E2 -6990.258} C_VEL
LIN {X 0,Y 481.694,Z 464.478,A -85,B 0,C 180,E1 -6993.109,E2 -6993.109} C_VEL
LIN {X 0,Y 481.638,Z 464.487,A -85,B 0,C 180,E1 -6995.885,E2 -6995.885} C_VEL
LIN {X 0,Y 481.689,Z 464.48,A -85,B 0,C 180,E1 -6999.027,E2 -6999.027} C_VEL
LIN {X 0,Y 481.689,Z 464.483,A -85,B 0,C 180,E1 -7002.157,E2 -7002.157} C_VEL
LIN {X 0,Y 481.728,Z 464.478,A -85,B 0,C 180,E1 -7004.775,E2 -7004.775} C_VEL
LIN {X 0,Y 481.739,Z 464.477,A -85,B 0,C 180,E1 -7008.214,E2 -7008.214} C_VEL
LIN {X 0,Y 481.748,Z 464.471,A -85,B 0,C 180,E1 -7011.611,E2 -7011.611} C_VEL
LIN {X 0,Y 481.79,Z 464.47,A -85,B 0,C 180,E1 -7014.139,E2 -7014.139} C_VEL
LIN {X 0,Y 481.912,Z 464.451,A -85,B 0,C 180,E1 -7017.492,E2 -7017.492} C_VEL
LIN {X 0,Y 481.912,Z 464.456,A -85,B 0,C 180,E1 -7020.835,E2 -7020.835} C_VEL
LIN {X 0,Y 481.913,Z 464.459,A -85,B 0,C 180,E1 -7022.507,E2 -7022.507} C_VEL
LIN {X 0,Y 481.794,Z 464.466,A -85,B 0,C 180,E1 -7025.86,E2 -7025.86} C_VEL
LIN {X 0,Y 481.75,Z 464.477,A -85,B 0,C 180,E1 -7028.388,E2 -7028.388} C_VEL
LIN {X 0,Y 481.738,Z 464.473,A -85,B 0,C 180,E1 -7031.785,E2 -7031.785} C_VEL
LIN {X 0,Y 481.73,Z 464.475,A -85,B 0,C 180,E1 -7035.224,E2 -7035.224} C_VEL
LIN {X 0,Y 481.698,Z 464.486,A -85,B 0,C 180,E1 -7038.722,E2 -7038.722} C_VEL
LIN {X 0,Y 481.633,Z 464.486,A -85,B 0,C 180,E1 -7041.395,E2 -7041.395} C_VEL
LIN {X 0,Y 481.663,Z 464.483,A -85,B 0,C 180,E1 -7044.114,E2 -7044.114} C_VEL
LIN {X 0,Y 481.738,Z 464.476,A -85,B 0,C 180,E1 -7047.141,E2 -7047.141} C_VEL
LIN {X 0,Y 481.665,Z 464.481,A -85,B 0,C 180,E1 -7049.742,E2 -7049.742} C_VEL
LIN {X 0,Y 481.66,Z 464.489,A -85,B 0,C 180,E1 -7052.675,E2 -7052.675} C_VEL
LIN {X 0,Y 481.63,Z 464.486,A -85,B 0,C 180,E1 -7055.71,E2 -7055.71} C_VEL
LIN {X 0,Y 481.659,Z 464.491,A -85,B 0,C 180,E1 -7058.86,E2 -7058.86} C_VEL
LIN {X 0,Y 481.65,Z 464.483,A -85,B 0,C 180,E1 -7061.915,E2 -7061.915} C_VEL
LIN {X 0,Y 481.648,Z 464.487,A -85,B 0,C 180,E1 -7064.458,E2 -7064.458} C_VEL
LIN {X 0,Y 481.678,Z 464.488,A -85,B 0,C 180,E1 -7066.847,E2 -7066.847} C_VEL
LIN {X 0,Y 481.683,Z 464.479,A -85,B 0,C 180,E1 -7070.062,E2 -7070.062} C_VEL
LIN {X 0,Y 481.619,Z 464.492,A -85,B 0,C 180,E1 -7073.255,E2 -7073.255} C_VEL
LIN {X 0,Y 481.7,Z 464.478,A -85,B 0,C 180,E1 -7076.331,E2 -7076.331} C_VEL
LIN {X 0,Y 481.643,Z 464.487,A -85,B 0,C 180,E1 -7079.418,E2 -7079.418} C_VEL
LIN {X 0,Y 481.693,Z 464.478,A -85,B 0,C 180,E1 -7082.169,E2 -7082.169} C_VEL
LIN {X 0,Y 481.711,Z 464.484,A -85,B 0,C 180,E1 -7084.971,E2 -7084.971} C_VEL
LIN {X 0,Y 481.63,Z 464.486,A -85,B 0,C 180,E1 -7087.999,E2 -7087.999} C_VEL
LIN {X 0,Y 480.964,Z 464.574,A -85,B 0,C 180,E1 -7088.697,E2 -7088.697} C_VEL
LIN {X 0,Y 478.136,Z 464.925,A -85,B 0,C 180,E1 -7089.831,E2 -7089.831} C_VEL
LIN {X 0,Y 475.751,Z 465.223,A -85,B 0,C 180,E1 -7090.745,E2 -7090.745} C_VEL
LIN {X 0,Y 474.731,Z 465.349,A -85,B 0,C 180,E1 -7091.451,E2 -7091.451} C_VEL
LIN {X 0,Y 474.65,Z 465.357,A -85,B 0,C 180,E1 -7091.69,E2 -7091.69} C_VEL
LIN {X 0,Y 474.695,Z 465.352,A -85,B 0,C 180,E1 -7094.546,E2 -7094.546} C_VEL
LIN {X 0,Y 474.7,Z 465.349,A -85,B 0,C 180,E1 -7098.039,E2 -7098.039} C_VEL
LIN {X 0,Y 474.726,Z 465.352,A -85,B 0,C 180,E1 -7101.488,E2 -7101.488} C_VEL
LIN {X 0,Y 474.779,Z 465.344,A -85,B 0,C 180,E1 -7104.054,E2 -7104.054} C_VEL
LIN {X 0,Y 474.895,Z 465.445,A -85,B 0,C 180,E1 -7107.613,E2 -7107.613} C_VEL
LIN {X 0,Y 475.05,Z 466.414,A -85,B 0,C 180,E1 -7107.769,E2 -7107.769} C_VEL
LIN {X 0,Y 478.154,Z 475.58,A -85,B 0,C 180,E1 -7108.034,E2 -7108.034} C_VEL
LIN {X 0,Y 477.732,Z 545.653,A -85,B 0,C 180,E1 -7109.106,E2 -7109.106} C_VEL
LIN {X 0,Y 477.654,Z 558.197,A -85,B 0,C 180,E1 -7109.448,E2 -7109.448} C_VEL
LIN {X 0,Y 477.507,Z 570.442,A -85,B 0,C 180,E1 -7109.949,E2 -7109.949} C_VEL
LIN {X 0,Y 477.198,Z 582.824,A -85,B 0,C 180,E1 -7110.634,E2 -7110.634} C_VEL
LIN {X 0,Y 476.839,Z 594.407,A -85,B 0,C 180,E1 -7111.479,E2 -7111.479} C_VEL
LIN {X 0,Y 476.41,Z 604.799,A -85,B 0,C 180,E1 -7112.432,E2 -7112.432} C_VEL
LIN {X 0,Y 476.021,Z 614.992,A -85,B 0,C 180,E1 -7113.599,E2 -7113.599} C_VEL
LIN {X 0,Y 475.627,Z 623.855,A -85,B 0,C 180,E1 -7114.875,E2 -7114.875} C_VEL
LIN {X 0,Y 475.332,Z 631.003,A -85,B 0,C 180,E1 -7116.155,E2 -7116.155} C_VEL
LIN {X 0,Y 475.02,Z 637.275,A -85,B 0,C 180,E1 -7117.577,E2 -7117.577} C_VEL
LIN {X 0,Y 474.79,Z 641.898,A -85,B 0,C 180,E1 -7118.943,E2 -7118.943} C_VEL
LIN {X 0,Y 474.588,Z 645.185,A -85,B 0,C 180,E1 -7120.237,E2 -7120.237} C_VEL
LIN {X 0,Y 474.508,Z 646.817,A -85,B 0,C 180,E1 -7121.103,E2 -7121.103} C_VEL
LIN {X 0,Y 474.481,Z 648.241,A -85,B 0,C 180,E1 -7122.154,E2 -7122.154} C_VEL
LIN {X 0,Y 474.419,Z 649.226,A -85,B 0,C 180,E1 -7123.712,E2 -7123.712} C_VEL
LIN {X 0,Y 474.409,Z 649.225,A -85,B 0,C 180,E1 -7124.588,E2 -7124.588} C_VEL
LIN {X 0,Y 474.473,Z 648.629,A -85,B 0,C 180,E1 -7125.679,E2 -7125.679} C_VEL
LIN {X 0,Y 474.593,Z 646.68,A -85,B 0,C 180,E1 -7127.229,E2 -7127.229} C_VEL
LIN {X 0,Y 474.776,Z 643.656,A -85,B 0,C 180,E1 -7128.671,E2 -7128.671} C_VEL
LIN {X 0,Y 474.975,Z 640.067,A -85,B 0,C 180,E1 -7129.898,E2 -7129.898} C_VEL
LIN {X 0,Y 475.27,Z 634.678,A -85,B 0,C 180,E1 -7131.314,E2 -7131.314} C_VEL
LIN {X 0,Y 475.586,Z 628.424,A -85,B 0,C 180,E1 -7132.596,E2 -7132.596} C_VEL
LIN {X 0,Y 475.948,Z 621.667,A -85,B 0,C 180,E1 -7133.722,E2 -7133.722} C_VEL
LIN {X 0,Y 476.367,Z 613.285,A -85,B 0,C 180,E1 -7134.866,E2 -7134.866} C_VEL
LIN {X 0,Y 476.772,Z 603.54,A -85,B 0,C 180,E1 -7135.949,E2 -7135.949} C_VEL
LIN {X 0,Y 477.161,Z 593.938,A -85,B 0,C 180,E1 -7136.814,E2 -7136.814} C_VEL
LIN {X 0,Y 477.557,Z 582.947,A -85,B 0,C 180,E1 -7137.605,E2 -7137.605} C_VEL
LIN {X 0,Y 477.871,Z 570.078,A -85,B 0,C 180,E1 -7138.315,E2 -7138.315} C_VEL
LIN {X 0,Y 477.965,Z 557.552,A -85,B 0,C 180,E1 -7138.818,E2 -7138.818} C_VEL
LIN {X 0,Y 478.063,Z 543.982,A -85,B 0,C 180,E1 -7139.16,E2 -7139.16} C_VEL
LIN {X 0,Y 478.431,Z 475.782,A -85,B 0,C 180,E1 -7140.219,E2 -7140.219} C_VEL
LIN {X 0,Y 474.787,Z 466.229,A -85,B 0,C 180,E1 -7140.546,E2 -7140.546} C_VEL
LIN {X 0,Y 474.616,Z 465.459,A -85,B 0,C 180,E1 -7140.702,E2 -7140.702} C_VEL
LIN {X 0,Y 474.628,Z 465.363,A -85,B 0,C 180,E1 -7143.223,E2 -7143.223} C_VEL
LIN {X 0,Y 474.592,Z 465.369,A -85,B 0,C 180,E1 -7146.325,E2 -7146.325} C_VEL
LIN {X 0,Y 474.622,Z 465.359,A -85,B 0,C 180,E1 -7149.647,E2 -7149.647} C_VEL
LIN {X 0,Y 474.628,Z 465.36,A -85,B 0,C 180,E1 -7152.238,E2 -7152.238} C_VEL
LIN {X 0,Y 474.621,Z 465.364,A -85,B 0,C 180,E1 -7155.299,E2 -7155.299} C_VEL
LIN {X 0,Y 474.625,Z 465.364,A -85,B 0,C 180,E1 -7158.216,E2 -7158.216} C_VEL
LIN {X 0,Y 474.675,Z 465.462,A -85,B 0,C 180,E1 -7161.633,E2 -7161.633} C_VEL
LIN {X 0,Y 476.937,Z 476.877,A -85,B 0,C 180,E1 -7163.622,E2 -7163.622} C_VEL
LIN {X 0,Y 476.672,Z 491.227,A -85,B 0,C 180,E1 -7165.926,E2 -7165.926} C_VEL
LIN {X 0,Y 476.131,Z 509.667,A -85,B 0,C 180,E1 -7168.894,E2 -7168.894} C_VEL
LIN {X 0,Y 475.924,Z 518.671,A -85,B 0,C 180,E1 -7170.316,E2 -7170.316} C_VEL
LIN {X 0,Y 478.095,Z 531.915,A -85,B 0,C 180,E1 -7170.642,E2 -7170.642} C_VEL
LIN {X 0,Y 477.232,Z 627.613,A -85,B 0,C 180,E1 -7172.194,E2 -7172.194} C_VEL
LIN {X 0,Y 476.946,Z 640.534,A -85,B 0,C 180,E1 -7172.561,E2 -7172.561} C_VEL
LIN {X 0,Y 476.549,Z 653.011,A -85,B 0,C 180,E1 -7173.092,E2 -7173.092} C_VEL
LIN {X 0,Y 476.223,Z 665.364,A -85,B 0,C 180,E1 -7173.804,E2 -7173.804} C_VEL
LIN {X 0,Y 475.813,Z 676.577,A -85,B 0,C 180,E1 -7174.638,E2 -7174.638} C_VEL
LIN {X 0,Y 475.286,Z 687.482,A -85,B 0,C 180,E1 -7175.658,E2 -7175.658} C_VEL
LIN {X 0,Y 474.933,Z 697.147,A -85,B 0,C 180,E1 -7176.783,E2 -7176.783} C_VEL
LIN {X 0,Y 474.537,Z 705.823,A -85,B 0,C 180,E1 -7178.04,E2 -7178.04} C_VEL
LIN {X 0,Y 474.262,Z 713.322,A -85,B 0,C 180,E1 -7179.394,E2 -7179.394} C_VEL
LIN {X 0,Y 474.1,Z 718.303,A -85,B 0,C 180,E1 -7180.517,E2 -7180.517} C_VEL
LIN {X 0,Y 473.935,Z 723.033,A -85,B 0,C 180,E1 -7181.856,E2 -7181.856} C_VEL
LIN {X 0,Y 473.828,Z 725.476,A -85,B 0,C 180,E1 -7182.744,E2 -7182.744} C_VEL
LIN {X 0,Y 473.772,Z 727.459,A -85,B 0,C 180,E1 -7183.63,E2 -7183.63} C_VEL
LIN {X 0,Y 473.715,Z 729.144,A -85,B 0,C 180,E1 -7184.655,E2 -7184.655} C_VEL
LIN {X 0,Y 473.673,Z 730.619,A -85,B 0,C 180,E1 -7186.267,E2 -7186.267} C_VEL
LIN {X 0,Y 473.685,Z 730.804,A -85,B 0,C 180,E1 -7187.141,E2 -7187.141} C_VEL
LIN {X 0,Y 473.784,Z 730.418,A -85,B 0,C 180,E1 -7188.249,E2 -7188.249} C_VEL
LIN {X 0,Y 473.78,Z 728.822,A -85,B 0,C 180,E1 -7189.747,E2 -7189.747} C_VEL
LIN {X 0,Y 473.81,Z 727.292,A -85,B 0,C 180,E1 -7190.61,E2 -7190.61} C_VEL
LIN {X 0,Y 473.961,Z 724.184,A -85,B 0,C 180,E1 -7191.902,E2 -7191.902} C_VEL
LIN {X 0,Y 474.1,Z 719.523,A -85,B 0,C 180,E1 -7193.322,E2 -7193.322} C_VEL
LIN {X 0,Y 474.287,Z 713.664,A -85,B 0,C 180,E1 -7194.686,E2 -7194.686} C_VEL
LIN {X 0,Y 474.523,Z 706.68,A -85,B 0,C 180,E1 -7195.966,E2 -7195.966} C_VEL
LIN {X 0,Y 474.893,Z 698.012,A -85,B 0,C 180,E1 -7197.243,E2 -7197.243} C_VEL
LIN {X 0,Y 475.276,Z 689.103,A -85,B 0,C 180,E1 -7198.306,E2 -7198.306} C_VEL
LIN {X 0,Y 475.759,Z 678.006,A -85,B 0,C 180,E1 -7199.366,E2 -7199.366} C_VEL
LIN {X 0,Y 476.164,Z 666.912,A -85,B 0,C 180,E1 -7200.212,E2 -7200.212} C_VEL
LIN {X 0,Y 476.618,Z 654.233,A -85,B 0,C 180,E1 -7200.951,E2 -7200.951} C_VEL
LIN {X 0,Y 476.967,Z 642.106,A -85,B 0,C 180,E1 -7201.478,E2 -7201.478} C_VEL
LIN {X 0,Y 477.176,Z 629.792,A -85,B 0,C 180,E1 -7201.847,E2 -7201.847} C_VEL
LIN {X 0,Y 477.519,Z 593.972,A -85,B 0,C 180,E1 -7202.452,E2 -7202.452} C_VEL
LIN {X 0,Y 478.151,Z 531.486,A -85,B 0,C 180,E1 -7203.489,E2 -7203.489} C_VEL
LIN {X 0,Y 476.166,Z 520.042,A -85,B 0,C 180,E1 -7203.782,E2 -7203.782} C_VEL
LIN {X 0,Y 476.495,Z 502.164,A -85,B 0,C 180,E1 -7206.564,E2 -7206.564} C_VEL
LIN {X 0,Y 476.89,Z 485.953,A -85,B 0,C 180,E1 -7209.103,E2 -7209.103} C_VEL
LIN {X 0,Y 477.012,Z 477.505,A -85,B 0,C 180,E1 -7210.398,E2 -7210.398} C_VEL
LIN {X 0,Y 475.068,Z 467.022,A -85,B 0,C 180,E1 -7212.113,E2 -7212.113} C_VEL
LIN {X 0,Y 474.695,Z 465.417,A -85,B 0,C 180,E1 -7212.442,E2 -7212.442} C_VEL
LIN {X 0,Y 474.688,Z 465.357,A -85,B 0,C 180,E1 -7215.767,E2 -7215.767} C_VEL
LIN {X 0,Y 474.67,Z 465.361,A -85,B 0,C 180,E1 -7219.01,E2 -7219.01} C_VEL
LIN {X 0,Y 474.596,Z 465.366,A -85,B 0,C 180,E1 -7221.729,E2 -7221.729} C_VEL
LIN {X 0,Y 474.637,Z 465.363,A -85,B 0,C 180,E1 -7224.494,E2 -7224.494} C_VEL
LIN {X 0,Y 474.682,Z 465.357,A -85,B 0,C 180,E1 -7227.332,E2 -7227.332} C_VEL
LIN {X 0,Y 474.613,Z 465.364,A -85,B 0,C 180,E1 -7230.23,E2 -7230.23} C_VEL
LIN {X 0,Y 474.651,Z 465.359,A -85,B 0,C 180,E1 -7233.22,E2 -7233.22} C_VEL
LIN {X 0,Y 474.597,Z 465.367,A -85,B 0,C 180,E1 -7236.323,E2 -7236.323} C_VEL
LIN {X 0,Y 474.626,Z 465.361,A -85,B 0,C 180,E1 -7239.646,E2 -7239.646} C_VEL
LIN {X 0,Y 474.622,Z 465.364,A -85,B 0,C 180,E1 -7242.934,E2 -7242.934} C_VEL
LIN {X 0,Y 474.614,Z 465.365,A -85,B 0,C 180,E1 -7245.894,E2 -7245.894} C_VEL
LIN {X 0,Y 474.635,Z 465.361,A -85,B 0,C 180,E1 -7249.04,E2 -7249.04} C_VEL
LIN {X 0,Y 474.614,Z 465.351,A -85,B 0,C 180,E1 -7251.704,E2 -7251.704} C_VEL
LIN {X 0,Y 474.626,Z 465.358,A -85,B 0,C 180,E1 -7254.724,E2 -7254.724} C_VEL
LIN {X 0,Y 474.635,Z 465.364,A -85,B 0,C 180,E1 -7257.786,E2 -7257.786} C_VEL
LIN {X 0,Y 474.683,Z 465.498,A -85,B 0,C 180,E1 -7259.774,E2 -7259.774} C_VEL
LIN {X 0,Y 477.41,Z 477.504,A -85,B 0,C 180,E1 -7261.655,E2 -7261.655} C_VEL
LIN {X 0,Y 478.405,Z 482.769,A -85,B 0,C 180,E1 -7262.434,E2 -7262.434} C_VEL
LIN {X 0,Y 477.434,Z 506.805,A -85,B 0,C 180,E1 -7265.657,E2 -7265.657} C_VEL
LIN {X 0,Y 476.555,Z 529.182,A -85,B 0,C 180,E1 -7268.591,E2 -7268.591} C_VEL
LIN {X 0,Y 475.666,Z 554.994,A -85,B 0,C 180,E1 -7271.923,E2 -7271.923} C_VEL
LIN {X 0,Y 475.392,Z 564.94,A -85,B 0,C 180,E1 -7273.175,E2 -7273.175} C_VEL
LIN {X 0,Y 477.89,Z 588.793,A -85,B 0,C 180,E1 -7273.655,E2 -7273.655} C_VEL
LIN {X 0,Y 477.28,Z 675.557,A -85,B 0,C 180,E1 -7274.984,E2 -7274.984} C_VEL
LIN {X 0,Y 476.874,Z 688.927,A -85,B 0,C 180,E1 -7275.353,E2 -7275.353} C_VEL
LIN {X 0,Y 476.391,Z 702.34,A -85,B 0,C 180,E1 -7275.91,E2 -7275.91} C_VEL
LIN {X 0,Y 475.934,Z 713.637,A -85,B 0,C 180,E1 -7276.55,E2 -7276.55} C_VEL
LIN {X 0,Y 475.433,Z 725.108,A -85,B 0,C 180,E1 -7277.381,E2 -7277.381} C_VEL
LIN {X 0,Y 475.032,Z 734.934,A -85,B 0,C 180,E1 -7278.261,E2 -7278.261} C_VEL
LIN {X 0,Y 474.605,Z 746.745,A -85,B 0,C 180,E1 -7279.547,E2 -7279.547} C_VEL
LIN {X 0,Y 474.362,Z 754.91,A -85,B 0,C 180,E1 -7280.619,E2 -7280.619} C_VEL
LIN {X 0,Y 474.142,Z 762.873,A -85,B 0,C 180,E1 -7281.904,E2 -7281.904} C_VEL
LIN {X 0,Y 473.984,Z 769.223,A -85,B 0,C 180,E1 -7283.186,E2 -7283.186} C_VEL
LIN {X 0,Y 473.976,Z 774.252,A -85,B 0,C 180,E1 -7284.468,E2 -7284.468} C_VEL
LIN {X 0,Y 473.922,Z 778.091,A -85,B 0,C 180,E1 -7285.746,E2 -7285.746} C_VEL
LIN {X 0,Y 473.924,Z 780.068,A -85,B 0,C 180,E1 -7286.598,E2 -7286.598} C_VEL
LIN {X 0,Y 473.907,Z 781.571,A -85,B 0,C 180,E1 -7287.449,E2 -7287.449} C_VEL
LIN {X 0,Y 473.862,Z 782.629,A -85,B 0,C 180,E1 -7288.299,E2 -7288.299} C_VEL
LIN {X 0,Y 473.821,Z 783.28,A -85,B 0,C 180,E1 -7289.149,E2 -7289.149} C_VEL
LIN {X 0,Y 473.868,Z 783.525,A -85,B 0,C 180,E1 -7289.999,E2 -7289.999} C_VEL
LIN {X 0,Y 473.818,Z 783.314,A -85,B 0,C 180,E1 -7290.848,E2 -7290.848} C_VEL
LIN {X 0,Y 473.857,Z 782.698,A -85,B 0,C 180,E1 -7291.698,E2 -7291.698} C_VEL
LIN {X 0,Y 473.901,Z 781.672,A -85,B 0,C 180,E1 -7292.549,E2 -7292.549} C_VEL
LIN {X 0,Y 473.915,Z 780.2,A -85,B 0,C 180,E1 -7293.399,E2 -7293.399} C_VEL
LIN {X 0,Y 473.874,Z 777.132,A -85,B 0,C 180,E1 -7294.677,E2 -7294.677} C_VEL
LIN {X 0,Y 473.957,Z 772.977,A -85,B 0,C 180,E1 -7295.956,E2 -7295.956} C_VEL
LIN {X 0,Y 474.026,Z 766.573,A -85,B 0,C 180,E1 -7297.452,E2 -7297.452} C_VEL
LIN {X 0,Y 474.225,Z 759.557,A -85,B 0,C 180,E1 -7298.736,E2 -7298.736} C_VEL
LIN {X 0,Y 474.474,Z 750.717,A -85,B 0,C 180,E1 -7300.021,E2 -7300.021} C_VEL
LIN {X 0,Y 474.859,Z 740.624,A -85,B 0,C 180,E1 -7301.199,E2 -7301.199} C_VEL
LIN {X 0,Y 475.408,Z 728.035,A -85,B 0,C 180,E1 -7302.397,E2 -7302.397} C_VEL
LIN {X 0,Y 475.771,Z 717.094,A -85,B 0,C 180,E1 -7303.234,E2 -7303.234} C_VEL
LIN {X 0,Y 476.301,Z 704.615,A -85,B 0,C 180,E1 -7303.981,E2 -7303.981} C_VEL
LIN {X 0,Y 476.732,Z 692.806,A -85,B 0,C 180,E1 -7304.512,E2 -7304.512} C_VEL
LIN {X 0,Y 477.181,Z 680.16,A -85,B 0,C 180,E1 -7304.907,E2 -7304.907} C_VEL
LIN {X 0,Y 477.367,Z 664.069,A -85,B 0,C 180,E1 -7305.202,E2 -7305.202} C_VEL
LIN {X 0,Y 477.752,Z 586.673,A -85,B 0,C 180,E1 -7306.373,E2 -7306.373} C_VEL
LIN {X 0,Y 475.407,Z 565.713,A -85,B 0,C 180,E1 -7306.781,E2 -7306.781} C_VEL
LIN {X 0,Y 476.084,Z 543.32,A -85,B 0,C 180,E1 -7309.622,E2 -7309.622} C_VEL
LIN {X 0,Y 476.93,Z 519.082,A -85,B 0,C 180,E1 -7312.755,E2 -7312.755} C_VEL
LIN {X 0,Y 477.743,Z 496.46,A -85,B 0,C 180,E1 -7315.718,E2 -7315.718} C_VEL
LIN {X 0,Y 478.283,Z 482.479,A -85,B 0,C 180,E1 -7317.57,E2 -7317.57} C_VEL
LIN {X 0,Y 474.78,Z 466.092,A -85,B 0,C 180,E1 -7319.977,E2 -7319.977} C_VEL
LIN {X 0,Y 474.673,Z 465.477,A -85,B 0,C 180,E1 -7320.104,E2 -7320.104} C_VEL
LIN {X 0,Y 474.619,Z 465.364,A -85,B 0,C 180,E1 -7323.22,E2 -7323.22} C_VEL
LIN {X 0,Y 474.574,Z 465.371,A -85,B 0,C 180,E1 -7326.323,E2 -7326.323} C_VEL
LIN {X 0,Y 474.593,Z 465.365,A -85,B 0,C 180,E1 -7329.642,E2 -7329.642} C_VEL
LIN {X 0,Y 474.579,Z 465.373,A -85,B 0,C 180,E1 -7332.23,E2 -7332.23} C_VEL
LIN {X 0,Y 474.607,Z 465.361,A -85,B 0,C 180,E1 -7335.296,E2 -7335.296} C_VEL
LIN {X 0,Y 474.599,Z 465.37,A -85,B 0,C 180,E1 -7338.212,E2 -7338.212} C_VEL
LIN {X 0,Y 474.597,Z 465.363,A -85,B 0,C 180,E1 -7341.541,E2 -7341.541} C_VEL
LIN {X 0,Y 474.611,Z 465.363,A -85,B 0,C 180,E1 -7344.724,E2 -7344.724} C_VEL
LIN {X 0,Y 474.624,Z 465.361,A -85,B 0,C 180,E1 -7347.787,E2 -7347.787} C_VEL
LIN {X 0,Y 474.609,Z 465.362,A -85,B 0,C 180,E1 -7350.884,E2 -7350.884} C_VEL
LIN {X 0,Y 474.615,Z 465.36,A -85,B 0,C 180,E1 -7353.625,E2 -7353.625} C_VEL
LIN {X 0,Y 474.621,Z 465.364,A -85,B 0,C 180,E1 -7356.641,E2 -7356.641} C_VEL
LIN {X 0,Y 474.64,Z 465.361,A -85,B 0,C 180,E1 -7360.089,E2 -7360.089} C_VEL
LIN {X 0,Y 474.633,Z 465.361,A -85,B 0,C 180,E1 -7362.773,E2 -7362.773} C_VEL
LIN {X 0,Y 474.631,Z 465.358,A -85,B 0,C 180,E1 -7365.42,E2 -7365.42} C_VEL
LIN {X 0,Y 474.692,Z 465.353,A -85,B 0,C 180,E1 -7368.037,E2 -7368.037} C_VEL
LIN {X 0,Y 474.713,Z 465.347,A -85,B 0,C 180,E1 -7371.486,E2 -7371.486} C_VEL
LIN {X 0,Y 474.753,Z 465.345,A -85,B 0,C 180,E1 -7374.052,E2 -7374.052} C_VEL
LIN {X 0,Y 474.878,Z 465.327,A -85,B 0,C 180,E1 -7377.455,E2 -7377.455} C_VEL
LIN {X 0,Y 474.863,Z 465.333,A -85,B 0,C 180,E1 -7380.848,E2 -7380.848} C_VEL
LIN {X 0,Y 474.879,Z 465.336,A -85,B 0,C 180,E1 -7382.544,E2 -7382.544} C_VEL
LIN {X 0,Y 474.756,Z 465.343,A -85,B 0,C 180,E1 -7385.948,E2 -7385.948} C_VEL
LIN {X 0,Y 474.715,Z 465.355,A -85,B 0,C 180,E1 -7388.513,E2 -7388.513} C_VEL
LIN {X 0,Y 474.691,Z 465.351,A -85,B 0,C 180,E1 -7391.962,E2 -7391.962} C_VEL
LIN {X 0,Y 474.686,Z 465.351,A -85,B 0,C 180,E1 -7395.456,E2 -7395.456} C_VEL
LIN {X 0,Y 474.651,Z 465.359,A -85,B 0,C 180,E1 -7399.01,E2 -7399.01} C_VEL
LIN {X 0,Y 474.576,Z 465.365,A -85,B 0,C 180,E1 -7401.729,E2 -7401.729} C_VEL
LIN {X 0,Y 474.645,Z 465.361,A -85,B 0,C 180,E1 -7404.493,E2 -7404.493} C_VEL
LIN {X 0,Y 474.685,Z 465.353,A -85,B 0,C 180,E1 -7407.339,E2 -7407.339} C_VEL
LIN {X 0,Y 474.592,Z 465.371,A -85,B 0,C 180,E1 -7410.811,E2 -7410.811} C_VEL
LIN {X 0,Y 474.625,Z 465.359,A -85,B 0,C 180,E1 -7413.985,E2 -7413.985} C_VEL
LIN {X 0,Y 474.563,Z 465.374,A -85,B 0,C 180,E1 -7416.901,E2 -7416.901} C_VEL
LIN {X 0,Y 474.615,Z 465.36,A -85,B 0,C 180,E1 -7419.649,E2 -7419.649} C_VEL
LIN {X 0,Y 474.633,Z 465.365,A -85,B 0,C 180,E1 -7422.932,E2 -7422.932} C_VEL
LIN {X 0,Y 474.607,Z 465.361,A -85,B 0,C 180,E1 -7425.897,E2 -7425.897} C_VEL
LIN {X 0,Y 474.636,Z 465.364,A -85,B 0,C 180,E1 -7429.039,E2 -7429.039} C_VEL
LIN {X 0,Y 474.609,Z 465.361,A -85,B 0,C 180,E1 -7431.704,E2 -7431.704} C_VEL
LIN {X 0,Y 474.619,Z 465.365,A -85,B 0,C 180,E1 -7434.727,E2 -7434.727} C_VEL
LIN {X 0,Y 474.629,Z 465.358,A -85,B 0,C 180,E1 -7437.789,E2 -7437.789} C_VEL
LIN {X 0,Y 474.617,Z 465.367,A -85,B 0,C 180,E1 -7440.886,E2 -7440.886} C_VEL
LIN {X 0,Y 474.653,Z 465.356,A -85,B 0,C 180,E1 -7443.63,E2 -7443.63} C_VEL
LIN {X 0,Y 474.629,Z 465.361,A -85,B 0,C 180,E1 -7446.643,E2 -7446.643} C_VEL
LIN {X 0,Y 474.651,Z 465.355,A -85,B 0,C 180,E1 -7450.091,E2 -7450.091} C_VEL
LIN {X 0,Y 474.65,Z 465.357,A -85,B 0,C 180,E1 -7451.69,E2 -7451.69} C_VEL
LIN {X 0,Y 473.988,Z 465.439,A -85,B 0,C 180,E1 -7452.399,E2 -7452.399} C_VEL
LIN {X 0,Y 471.137,Z 465.799,A -85,B 0,C 180,E1 -7453.55,E2 -7453.55} C_VEL
LIN {X 0,Y 468.721,Z 466.103,A -85,B 0,C 180,E1 -7454.479,E2 -7454.479} C_VEL
LIN {X 0,Y 467.679,Z 466.231,A -85,B 0,C 180,E1 -7455.196,E2 -7455.196} C_VEL
LIN {X 0,Y 467.593,Z 466.238,A -85,B 0,C 180,E1 -7455.439,E2 -7455.439} C_VEL
LIN {X 0,Y 467.65,Z 466.231,A -85,B 0,C 180,E1 -7458.735,E2 -7458.735} C_VEL
LIN {X 0,Y 467.746,Z 466.219,A -85,B 0,C 180,E1 -7462.23,E2 -7462.23} C_VEL
LIN {X 0,Y 467.725,Z 466.224,A -85,B 0,C 180,E1 -7464.829,E2 -7464.829} C_VEL
LIN {X 0,Y 467.859,Z 466.401,A -85,B 0,C 180,E1 -7467.419,E2 -7467.419} C_VEL
LIN {X 0,Y 468.045,Z 467.164,A -85,B 0,C 180,E1 -7467.541,E2 -7467.541} C_VEL
LIN {X 0,Y 471.299,Z 477.288,A -85,B 0,C 180,E1 -7467.832,E2 -7467.832} C_VEL
LIN {X 0,Y 470.885,Z 546.649,A -85,B 0,C 180,E1 -7468.906,E2 -7468.906} C_VEL
LIN {X 0,Y 470.808,Z 559.174,A -85,B 0,C 180,E1 -7469.253,E2 -7469.253} C_VEL
LIN {X 0,Y 470.642,Z 571.971,A -85,B 0,C 180,E1 -7469.788,E2 -7469.788} C_VEL
LIN {X 0,Y 470.338,Z 583.368,A -85,B 0,C 180,E1 -7470.43,E2 -7470.43} C_VEL
LIN {X 0,Y 469.972,Z 595.059,A -85,B 0,C 180,E1 -7471.287,E2 -7471.287} C_VEL
LIN {X 0,Y 469.516,Z 605.508,A -85,B 0,C 180,E1 -7472.253,E2 -7472.253} C_VEL
LIN {X 0,Y 469.101,Z 615.763,A -85,B 0,C 180,E1 -7473.437,E2 -7473.437} C_VEL
LIN {X 0,Y 468.665,Z 624.667,A -85,B 0,C 180,E1 -7474.732,E2 -7474.732} C_VEL
LIN {X 0,Y 468.347,Z 631.846,A -85,B 0,C 180,E1 -7476.031,E2 -7476.031} C_VEL
LIN {X 0,Y 468.066,Z 637.816,A -85,B 0,C 180,E1 -7477.385,E2 -7477.385} C_VEL
LIN {X 0,Y 467.813,Z 642.173,A -85,B 0,C 180,E1 -7478.642,E2 -7478.642} C_VEL
LIN {X 0,Y 467.666,Z 644.584,A -85,B 0,C 180,E1 -7479.516,E2 -7479.516} C_VEL
LIN {X 0,Y 467.554,Z 646.557,A -85,B 0,C 180,E1 -7480.393,E2 -7480.393} C_VEL
LIN {X 0,Y 467.485,Z 648.117,A -85,B 0,C 180,E1 -7481.272,E2 -7481.272} C_VEL
LIN {X 0,Y 467.462,Z 649.318,A -85,B 0,C 180,E1 -7482.251,E2 -7482.251} C_VEL
LIN {X 0,Y 467.407,Z 650.25,A -85,B 0,C 180,E1 -7483.922,E2 -7483.922} C_VEL
LIN {X 0,Y 467.394,Z 650.172,A -85,B 0,C 180,E1 -7484.812,E2 -7484.812} C_VEL
LIN {X 0,Y 467.452,Z 649.55,A -85,B 0,C 180,E1 -7485.801,E2 -7485.801} C_VEL
LIN {X 0,Y 467.6,Z 647.353,A -85,B 0,C 180,E1 -7487.495,E2 -7487.495} C_VEL
LIN {X 0,Y 467.793,Z 644.488,A -85,B 0,C 180,E1 -7488.828,E2 -7488.828} C_VEL
LIN {X 0,Y 468.055,Z 640.414,A -85,B 0,C 180,E1 -7490.205,E2 -7490.205} C_VEL
LIN {X 0,Y 468.364,Z 634.525,A -85,B 0,C 180,E1 -7491.7,E2 -7491.7} C_VEL
LIN {X 0,Y 468.802,Z 627.032,A -85,B 0,C 180,E1 -7493.175,E2 -7493.175} C_VEL
LIN {X 0,Y 469.214,Z 620.035,A -85,B 0,C 180,E1 -7494.279,E2 -7494.279} C_VEL
LIN {X 0,Y 469.677,Z 610.673,A -85,B 0,C 180,E1 -7495.482,E2 -7495.482} C_VEL
LIN {X 0,Y 470.07,Z 600.907,A -85,B 0,C 180,E1 -7496.499,E2 -7496.499} C_VEL
LIN {X 0,Y 470.539,Z 590.869,A -85,B 0,C 180,E1 -7497.342,E2 -7497.342} C_VEL
LIN {X 0,Y 470.89,Z 580.545,A -85,B 0,C 180,E1 -7498.041,E2 -7498.041} C_VEL
LIN {X 0,Y 471.136,Z 567.894,A -85,B 0,C 180,E1 -7498.696,E2 -7498.696} C_VEL
LIN {X 0,Y 471.279,Z 555.262,A -85,B 0,C 180,E1 -7499.16,E2 -7499.16} C_VEL
LIN {X 0,Y 471.34,Z 541.966,A -85,B 0,C 180,E1 -7499.462,E2 -7499.462} C_VEL
LIN {X 0,Y 471.777,Z 477.433,A -85,B 0,C 180,E1 -7500.467,E2 -7500.467} C_VEL
LIN {X 0,Y 467.797,Z 467.304,A -85,B 0,C 180,E1 -7500.816,E2 -7500.816} C_VEL
LIN {X 0,Y 467.589,Z 466.397,A -85,B 0,C 180,E1 -7500.963,E2 -7500.963} C_VEL
LIN {X 0,Y 467.573,Z 466.242,A -85,B 0,C 180,E1 -7503.791,E2 -7503.791} C_VEL
LIN {X 0,Y 467.533,Z 466.246,A -85,B 0,C 180,E1 -7506.963,E2 -7506.963} C_VEL
LIN {X 0,Y 467.581,Z 466.235,A -85,B 0,C 180,E1 -7509.955,E2 -7509.955} C_VEL
LIN {X 0,Y 467.591,Z 466.236,A -85,B 0,C 180,E1 -7512.568,E2 -7512.568} C_VEL
LIN {X 0,Y 467.57,Z 466.245,A -85,B 0,C 180,E1 -7515.054,E2 -7515.054} C_VEL
LIN {X 0,Y 467.594,Z 466.24,A -85,B 0,C 180,E1 -7517.441,E2 -7517.441} C_VEL
LIN {X 0,Y 467.597,Z 466.243,A -85,B 0,C 180,E1 -7520.857,E2 -7520.857} C_VEL
LIN {X 0,Y 467.647,Z 466.416,A -85,B 0,C 180,E1 -7521.443,E2 -7521.443} C_VEL
LIN {X 0,Y 470.09,Z 478.841,A -85,B 0,C 180,E1 -7523.605,E2 -7523.605} C_VEL
LIN {X 0,Y 469.615,Z 496.987,A -85,B 0,C 180,E1 -7526.549,E2 -7526.549} C_VEL
LIN {X 0,Y 469.019,Z 517.511,A -85,B 0,C 180,E1 -7529.869,E2 -7529.869} C_VEL
LIN {X 0,Y 469.047,Z 519.073,A -85,B 0,C 180,E1 -7530.08,E2 -7530.08} C_VEL
LIN {X 0,Y 471.299,Z 533.414,A -85,B 0,C 180,E1 -7530.431,E2 -7530.431} C_VEL
LIN {X 0,Y 470.324,Z 628.586,A -85,B 0,C 180,E1 -7532.008,E2 -7532.008} C_VEL
LIN {X 0,Y 470.035,Z 641.393,A -85,B 0,C 180,E1 -7532.386,E2 -7532.386} C_VEL
LIN {X 0,Y 469.622,Z 654.455,A -85,B 0,C 180,E1 -7532.963,E2 -7532.963} C_VEL
LIN {X 0,Y 469.272,Z 666.094,A -85,B 0,C 180,E1 -7533.653,E2 -7533.653} C_VEL
LIN {X 0,Y 468.849,Z 676.904,A -85,B 0,C 180,E1 -7534.472,E2 -7534.472} C_VEL
LIN {X 0,Y 468.304,Z 687.824,A -85,B 0,C 180,E1 -7535.508,E2 -7535.508} C_VEL
LIN {X 0,Y 467.933,Z 697.47,A -85,B 0,C 180,E1 -7536.645,E2 -7536.645} C_VEL
LIN {X 0,Y 467.508,Z 706.192,A -85,B 0,C 180,E1 -7537.925,E2 -7537.925} C_VEL
LIN {X 0,Y 467.212,Z 713.706,A -85,B 0,C 180,E1 -7539.299,E2 -7539.299} C_VEL
LIN {X 0,Y 467.004,Z 719.56,A -85,B 0,C 180,E1 -7540.666,E2 -7540.666} C_VEL
LIN {X 0,Y 466.846,Z 724.073,A -85,B 0,C 180,E1 -7542.025,E2 -7542.025} C_VEL
LIN {X 0,Y 466.717,Z 727.399,A -85,B 0,C 180,E1 -7543.375,E2 -7543.375} C_VEL
LIN {X 0,Y 466.644,Z 729.44,A -85,B 0,C 180,E1 -7544.559,E2 -7544.559} C_VEL
LIN {X 0,Y 466.583,Z 730.893,A -85,B 0,C 180,E1 -7546.055,E2 -7546.055} C_VEL
LIN {X 0,Y 466.587,Z 731.197,A -85,B 0,C 180,E1 -7546.942,E2 -7546.942} C_VEL
LIN {X 0,Y 466.704,Z 730.859,A -85,B 0,C 180,E1 -7548.192,E2 -7548.192} C_VEL
LIN {X 0,Y 466.695,Z 729.499,A -85,B 0,C 180,E1 -7549.589,E2 -7549.589} C_VEL
LIN {X 0,Y 466.717,Z 728.094,A -85,B 0,C 180,E1 -7550.466,E2 -7550.466} C_VEL
LIN {X 0,Y 466.869,Z 725.135,A -85,B 0,C 180,E1 -7551.778,E2 -7551.778} C_VEL
LIN {X 0,Y 467.024,Z 720.261,A -85,B 0,C 180,E1 -7553.322,E2 -7553.322} C_VEL
LIN {X 0,Y 467.265,Z 713.934,A -85,B 0,C 180,E1 -7554.823,E2 -7554.823} C_VEL
LIN {X 0,Y 467.523,Z 706.906,A -85,B 0,C 180,E1 -7556.122,E2 -7556.122} C_VEL
LIN {X 0,Y 467.935,Z 698.186,A -85,B 0,C 180,E1 -7557.418,E2 -7557.418} C_VEL
LIN {X 0,Y 468.357,Z 688.177,A -85,B 0,C 180,E1 -7558.603,E2 -7558.603} C_VEL
LIN {X 0,Y 468.852,Z 678.037,A -85,B 0,C 180,E1 -7559.571,E2 -7559.571} C_VEL
LIN {X 0,Y 469.287,Z 666.844,A -85,B 0,C 180,E1 -7560.429,E2 -7560.429} C_VEL
LIN {X 0,Y 469.712,Z 655.112,A -85,B 0,C 180,E1 -7561.126,E2 -7561.126} C_VEL
LIN {X 0,Y 470.08,Z 643.168,A -85,B 0,C 180,E1 -7561.66,E2 -7561.66} C_VEL
LIN {X 0,Y 470.302,Z 631.37,A -85,B 0,C 180,E1 -7562.034,E2 -7562.034} C_VEL
LIN {X 0,Y 470.532,Z 607.964,A -85,B 0,C 180,E1 -7562.461,E2 -7562.461} C_VEL
LIN {X 0,Y 471.377,Z 532.18,A -85,B 0,C 180,E1 -7563.74,E2 -7563.74} C_VEL
LIN {X 0,Y 469.292,Z 520.418,A -85,B 0,C 180,E1 -7564.053,E2 -7564.053} C_VEL
LIN {X 0,Y 469.808,Z 498.422,A -85,B 0,C 180,E1 -7567.522,E2 -7567.522} C_VEL
LIN {X 0,Y 470.179,Z 480.307,A -85,B 0,C 180,E1 -7570.333,E2 -7570.333} C_VEL
LIN {X 0,Y 469.232,Z 473.504,A -85,B 0,C 180,E1 -7571.447,E2 -7571.447} C_VEL
LIN {X 0,Y 467.629,Z 466.348,A -85,B 0,C 180,E1 -7572.677,E2 -7572.677} C_VEL
LIN {X 0,Y 467.657,Z 466.232,A -85,B 0,C 180,E1 -7575.885,E2 -7575.885} C_VEL
LIN {X 0,Y 467.629,Z 466.237,A -85,B 0,C 180,E1 -7579.308,E2 -7579.308} C_VEL
LIN {X 0,Y 467.542,Z 466.245,A -85,B 0,C 180,E1 -7582.074,E2 -7582.074} C_VEL
LIN {X 0,Y 467.578,Z 466.244,A -85,B 0,C 180,E1 -7584.889,E2 -7584.889} C_VEL
LIN {X 0,Y 467.624,Z 466.234,A -85,B 0,C 180,E1 -7587.769,E2 -7587.769} C_VEL
LIN {X 0,Y 467.576,Z 466.243,A -85,B 0,C 180,E1 -7591.044,E2 -7591.044} C_VEL
LIN {X 0,Y 467.597,Z 466.238,A -85,B 0,C 180,E1 -7594.242,E2 -7594.242} C_VEL
LIN {X 0,Y 467.556,Z 466.243,A -85,B 0,C 180,E1 -7597.186,E2 -7597.186} C_VEL
LIN {X 0,Y 467.583,Z 466.241,A -85,B 0,C 180,E1 -7600.264,E2 -7600.264} C_VEL
LIN {X 0,Y 467.595,Z 466.24,A -85,B 0,C 180,E1 -7602.566,E2 -7602.566} C_VEL
LIN {X 0,Y 467.574,Z 466.241,A -85,B 0,C 180,E1 -7605.052,E2 -7605.052} C_VEL
LIN {X 0,Y 467.597,Z 466.237,A -85,B 0,C 180,E1 -7607.439,E2 -7607.439} C_VEL
LIN {X 0,Y 467.566,Z 466.232,A -85,B 0,C 180,E1 -7610.852,E2 -7610.852} C_VEL
LIN {X 0,Y 467.563,Z 466.244,A -85,B 0,C 180,E1 -7614.261,E2 -7614.261} C_VEL
LIN {X 0,Y 467.581,Z 466.243,A -85,B 0,C 180,E1 -7617.322,E2 -7617.322} C_VEL
LIN {X 0,Y 467.631,Z 466.412,A -85,B 0,C 180,E1 -7619.504,E2 -7619.504} C_VEL
LIN {X 0,Y 470.444,Z 478.585,A -85,B 0,C 180,E1 -7621.44,E2 -7621.44} C_VEL
LIN {X 0,Y 471.534,Z 484.157,A -85,B 0,C 180,E1 -7622.285,E2 -7622.285} C_VEL
LIN {X 0,Y 470.635,Z 504.359,A -85,B 0,C 180,E1 -7625.047,E2 -7625.047} C_VEL
LIN {X 0,Y 469.61,Z 529.088,A -85,B 0,C 180,E1 -7628.357,E2 -7628.357} C_VEL
LIN {X 0,Y 468.693,Z 554.089,A -85,B 0,C 180,E1 -7631.644,E2 -7631.644} C_VEL
LIN {X 0,Y 468.407,Z 564.168,A -85,B 0,C 180,E1 -7632.919,E2 -7632.919} C_VEL
LIN {X 0,Y 471.071,Z 589.166,A -85,B 0,C 180,E1 -7633.424,E2 -7633.424} C_VEL
LIN {X 0,Y 470.388,Z 674.828,A -85,B 0,C 180,E1 -7634.758,E2 -7634.758} C_VEL
LIN {X 0,Y 469.961,Z 688.069,A -85,B 0,C 180,E1 -7635.133,E2 -7635.133} C_VEL
LIN {X 0,Y 469.492,Z 701.409,A -85,B 0,C 180,E1 -7635.699,E2 -7635.699} C_VEL
LIN {X 0,Y 468.962,Z 712.671,A -85,B 0,C 180,E1 -7636.346,E2 -7636.346} C_VEL
LIN {X 0,Y 468.394,Z 724.725,A -85,B 0,C 180,E1 -7637.238,E2 -7637.238} C_VEL
LIN {X 0,Y 467.973,Z 735.042,A -85,B 0,C 180,E1 -7638.191,E2 -7638.191} C_VEL
LIN {X 0,Y 467.644,Z 744.369,A -85,B 0,C 180,E1 -7639.171,E2 -7639.171} C_VEL
LIN {X 0,Y 467.334,Z 752.882,A -85,B 0,C 180,E1 -7640.258,E2 -7640.258} C_VEL
LIN {X 0,Y 467.121,Z 761.187,A -85,B 0,C 180,E1 -7641.563,E2 -7641.563} C_VEL
LIN {X 0,Y 466.945,Z 766.808,A -85,B 0,C 180,E1 -7642.648,E2 -7642.648} C_VEL
LIN {X 0,Y 466.868,Z 772.285,A -85,B 0,C 180,E1 -7643.95,E2 -7643.95} C_VEL
LIN {X 0,Y 466.812,Z 776.521,A -85,B 0,C 180,E1 -7645.249,E2 -7645.249} C_VEL
LIN {X 0,Y 466.851,Z 779.65,A -85,B 0,C 180,E1 -7646.546,E2 -7646.546} C_VEL
LIN {X 0,Y 466.818,Z 781.162,A -85,B 0,C 180,E1 -7647.41,E2 -7647.41} C_VEL
LIN {X 0,Y 466.792,Z 782.226,A -85,B 0,C 180,E1 -7648.273,E2 -7648.273} C_VEL
LIN {X 0,Y 466.744,Z 782.882,A -85,B 0,C 180,E1 -7649.136,E2 -7649.136} C_VEL
LIN {X 0,Y 466.785,Z 783.132,A -85,B 0,C 180,E1 -7649.999,E2 -7649.999} C_VEL
LIN {X 0,Y 466.741,Z 782.917,A -85,B 0,C 180,E1 -7650.861,E2 -7650.861} C_VEL
LIN {X 0,Y 466.787,Z 782.299,A -85,B 0,C 180,E1 -7651.724,E2 -7651.724} C_VEL
LIN {X 0,Y 466.812,Z 781.274,A -85,B 0,C 180,E1 -7652.587,E2 -7652.587} C_VEL
LIN {X 0,Y 466.841,Z 779.796,A -85,B 0,C 180,E1 -7653.451,E2 -7653.451} C_VEL
LIN {X 0,Y 466.795,Z 776.725,A -85,B 0,C 180,E1 -7654.748,E2 -7654.748} C_VEL
LIN {X 0,Y 466.856,Z 772.551,A -85,B 0,C 180,E1 -7656.047,E2 -7656.047} C_VEL
LIN {X 0,Y 466.953,Z 766.122,A -85,B 0,C 180,E1 -7657.566,E2 -7657.566} C_VEL
LIN {X 0,Y 467.142,Z 759.081,A -85,B 0,C 180,E1 -7658.869,E2 -7658.869} C_VEL
LIN {X 0,Y 467.436,Z 750.195,A -85,B 0,C 180,E1 -7660.174,E2 -7660.174} C_VEL
LIN {X 0,Y 467.817,Z 740.06,A -85,B 0,C 180,E1 -7661.37,E2 -7661.37} C_VEL
LIN {X 0,Y 468.328,Z 728.923,A -85,B 0,C 180,E1 -7662.417,E2 -7662.417} C_VEL
LIN {X 0,Y 468.732,Z 717.604,A -85,B 0,C 180,E1 -7663.327,E2 -7663.327} C_VEL
LIN {X 0,Y 469.289,Z 705.531,A -85,B 0,C 180,E1 -7664.083,E2 -7664.083} C_VEL
LIN {X 0,Y 469.784,Z 692.994,A -85,B 0,C 180,E1 -7664.676,E2 -7664.676} C_VEL
LIN {X 0,Y 470.287,Z 680.061,A -85,B 0,C 180,E1 -7665.103,E2 -7665.103} C_VEL
LIN {X 0,Y 470.465,Z 666.283,A -85,B 0,C 180,E1 -7665.375,E2 -7665.375} C_VEL
LIN {X 0,Y 470.923,Z 587.471,A -85,B 0,C 180,E1 -7666.582,E2 -7666.582} C_VEL
LIN {X 0,Y 468.388,Z 564.592,A -85,B 0,C 180,E1 -7667.04,E2 -7667.04} C_VEL
LIN {X 0,Y 469.152,Z 540.529,A -85,B 0,C 180,E1 -7670.152,E2 -7670.152} C_VEL
LIN {X 0,Y 469.978,Z 518.048,A -85,B 0,C 180,E1 -7673.111,E2 -7673.111} C_VEL
LIN {X 0,Y 470.89,Z 495.638,A -85,B 0,C 180,E1 -7676.09,E2 -7676.09} C_VEL
LIN {X 0,Y 471.359,Z 483.567,A -85,B 0,C 180,E1 -7677.719,E2 -7677.719} C_VEL
LIN {X 0,Y 467.635,Z 466.433,A -85,B 0,C 180,E1 -7680.29,E2 -7680.29} C_VEL
LIN {X 0,Y 467.574,Z 466.243,A -85,B 0,C 180,E1 -7682.757,E2 -7682.757} C_VEL
LIN {X 0,Y 467.542,Z 466.248,A -85,B 0,C 180,E1 -7685.888,E2 -7685.888} C_VEL
LIN {X 0,Y 467.536,Z 466.242,A -85,B 0,C 180,E1 -7689.147,E2 -7689.147} C_VEL
LIN {X 0,Y 467.556,Z 466.239,A -85,B 0,C 180,E1 -7691.403,E2 -7691.403} C_VEL
LIN {X 0,Y 467.556,Z 466.239,A -85,B 0,C 180,E1 -7695.051,E2 -7695.051} C_VEL
LIN {X 0,Y 467.557,Z 466.243,A -85,B 0,C 180,E1 -7698.595,E2 -7698.595} C_VEL
LIN {X 0,Y 467.551,Z 466.244,A -85,B 0,C 180,E1 -7701.954,E2 -7701.954} C_VEL
LIN {X 0,Y 467.551,Z 466.24,A -85,B 0,C 180,E1 -7705.166,E2 -7705.166} C_VEL
LIN {X 0,Y 467.571,Z 466.245,A -85,B 0,C 180,E1 -7708.259,E2 -7708.259} C_VEL
LIN {X 0,Y 467.561,Z 466.239,A -85,B 0,C 180,E1 -7711.249,E2 -7711.249} C_VEL
LIN {X 0,Y 467.575,Z 466.242,A -85,B 0,C 180,E1 -7714.158,E2 -7714.158} C_VEL
LIN {X 0,Y 467.562,Z 466.24,A -85,B 0,C 180,E1 -7716.995,E2 -7716.995} C_VEL
LIN {X 0,Y 467.609,Z 466.234,A -85,B 0,C 180,E1 -7719.776,E2 -7719.776} C_VEL
LIN {X 0,Y 467.592,Z 466.242,A -85,B 0,C 180,E1 -7722.506,E2 -7722.506} C_VEL
LIN {X 0,Y 467.59,Z 466.235,A -85,B 0,C 180,E1 -7725.196,E2 -7725.196} C_VEL
LIN {X 0,Y 467.643,Z 466.23,A -85,B 0,C 180,E1 -7727.854,E2 -7727.854} C_VEL
LIN {X 0,Y 467.667,Z 466.225,A -85,B 0,C 180,E1 -7731.357,E2 -7731.357} C_VEL
LIN {X 0,Y 467.717,Z 466.221,A -85,B 0,C 180,E1 -7733.962,E2 -7733.962} C_VEL
LIN {X 0,Y 467.844,Z 466.203,A -85,B 0,C 180,E1 -7737.417,E2 -7737.417} C_VEL
LIN {X 0,Y 467.866,Z 466.202,A -85,B 0,C 180,E1 -7740,E2 -7740} C_VEL
LIN {X 0,Y 467.844,Z 466.212,A -85,B 0,C 180,E1 -7742.583,E2 -7742.583} C_VEL
LIN {X 0,Y 467.72,Z 466.22,A -85,B 0,C 180,E1 -7746.037,E2 -7746.037} C_VEL
LIN {X 0,Y 467.668,Z 466.234,A -85,B 0,C 180,E1 -7748.643,E2 -7748.643} C_VEL
LIN {X 0,Y 467.642,Z 466.231,A -85,B 0,C 180,E1 -7752.145,E2 -7752.145} C_VEL
LIN {X 0,Y 467.625,Z 466.231,A -85,B 0,C 180,E1 -7755.695,E2 -7755.695} C_VEL
LIN {X 0,Y 467.603,Z 466.241,A -85,B 0,C 180,E1 -7758.765,E2 -7758.765} C_VEL
LIN {X 0,Y 467.567,Z 466.239,A -85,B 0,C 180,E1 -7761.269,E2 -7761.269} C_VEL
LIN {X 0,Y 467.559,Z 466.239,A -85,B 0,C 180,E1 -7763.944,E2 -7763.944} C_VEL
LIN {X 0,Y 467.614,Z 466.24,A -85,B 0,C 180,E1 -7766.8,E2 -7766.8} C_VEL
LIN {X 0,Y 467.541,Z 466.241,A -85,B 0,C 180,E1 -7769.739,E2 -7769.739} C_VEL
LIN {X 0,Y 467.57,Z 466.246,A -85,B 0,C 180,E1 -7772.759,E2 -7772.759} C_VEL
LIN {X 0,Y 467.544,Z 466.241,A -85,B 0,C 180,E1 -7775.89,E2 -7775.89} C_VEL
LIN {X 0,Y 467.57,Z 466.242,A -85,B 0,C 180,E1 -7779.146,E2 -7779.146} C_VEL
LIN {X 0,Y 467.574,Z 466.241,A -85,B 0,C 180,E1 -7782.568,E2 -7782.568} C_VEL
LIN {X 0,Y 467.559,Z 466.245,A -85,B 0,C 180,E1 -7785.054,E2 -7785.054} C_VEL
LIN {X 0,Y 467.613,Z 466.234,A -85,B 0,C 180,E1 -7787.445,E2 -7787.445} C_VEL
LIN {X 0,Y 467.609,Z 466.24,A -85,B 0,C 180,E1 -7790.86,E2 -7790.86} C_VEL
LIN {X 0,Y 467.553,Z 466.24,A -85,B 0,C 180,E1 -7794.262,E2 -7794.262} C_VEL
LIN {X 0,Y 467.573,Z 466.241,A -85,B 0,C 180,E1 -7797.322,E2 -7797.322} C_VEL
LIN {X 0,Y 467.563,Z 466.242,A -85,B 0,C 180,E1 -7800.669,E2 -7800.669} C_VEL
LIN {X 0,Y 467.609,Z 466.238,A -85,B 0,C 180,E1 -7803.201,E2 -7803.201} C_VEL
LIN {X 0,Y 467.586,Z 466.237,A -85,B 0,C 180,E1 -7806.469,E2 -7806.469} C_VEL
LIN {X 0,Y 467.618,Z 466.232,A -85,B 0,C 180,E1 -7809.779,E2 -7809.779} C_VEL
LIN {X 0,Y 467.604,Z 466.235,A -85,B 0,C 180,E1 -7812.508,E2 -7812.508} C_VEL
LIN {X 0,Y 467.593,Z 466.238,A -85,B 0,C 180,E1 -7815.439,E2 -7815.439} C_VEL
LIN {X 0,Y 466.923,Z 466.319,A -85,B 0,C 180,E1 -7816.158,E2 -7816.158} C_VEL
LIN {X 0,Y 464.079,Z 466.678,A -85,B 0,C 180,E1 -7817.326,E2 -7817.326} C_VEL
LIN {X 0,Y 461.68,Z 466.974,A -85,B 0,C 180,E1 -7818.269,E2 -7818.269} C_VEL
LIN {X 0,Y 460.655,Z 467.105,A -85,B 0,C 180,E1 -7818.996,E2 -7818.996} C_VEL
LIN {X 0,Y 460.574,Z 467.113,A -85,B 0,C 180,E1 -7819.243,E2 -7819.243} C_VEL
LIN {X 0,Y 460.718,Z 467.096,A -85,B 0,C 180,E1 -7822.539,E2 -7822.539} C_VEL
LIN {X 0,Y 460.697,Z 467.099,A -85,B 0,C 180,E1 -7824.75,E2 -7824.75} C_VEL
LIN {X 0,Y 460.745,Z 467.215,A -85,B 0,C 180,E1 -7827.16,E2 -7827.16} C_VEL
LIN {X 0,Y 460.961,Z 468.062,A -85,B 0,C 180,E1 -7827.312,E2 -7827.312} C_VEL
LIN {X 0,Y 464.464,Z 478.419,A -85,B 0,C 180,E1 -7827.616,E2 -7827.616} C_VEL
LIN {X 0,Y 464.009,Z 548.61,A -85,B 0,C 180,E1 -7828.727,E2 -7828.727} C_VEL
LIN {X 0,Y 463.898,Z 562.241,A -85,B 0,C 180,E1 -7829.133,E2 -7829.133} C_VEL
LIN {X 0,Y 463.727,Z 574.493,A -85,B 0,C 180,E1 -7829.676,E2 -7829.676} C_VEL
LIN {X 0,Y 463.451,Z 585.499,A -85,B 0,C 180,E1 -7830.327,E2 -7830.327} C_VEL
LIN {X 0,Y 463.05,Z 596.918,A -85,B 0,C 180,E1 -7831.197,E2 -7831.197} C_VEL
LIN {X 0,Y 462.552,Z 607.233,A -85,B 0,C 180,E1 -7832.178,E2 -7832.178} C_VEL
LIN {X 0,Y 462.175,Z 616.504,A -85,B 0,C 180,E1 -7833.27,E2 -7833.27} C_VEL
LIN {X 0,Y 461.733,Z 625.454,A -85,B 0,C 180,E1 -7834.585,E2 -7834.585} C_VEL
LIN {X 0,Y 461.366,Z 632.678,A -85,B 0,C 180,E1 -7835.903,E2 -7835.903} C_VEL
LIN {X 0,Y 461.113,Z 637.583,A -85,B 0,C 180,E1 -7837.005,E2 -7837.005} C_VEL
LIN {X 0,Y 460.859,Z 642.353,A -85,B 0,C 180,E1 -7838.331,E2 -7838.331} C_VEL
LIN {X 0,Y 460.64,Z 646.026,A -85,B 0,C 180,E1 -7839.663,E2 -7839.663} C_VEL
LIN {X 0,Y 460.53,Z 647.928,A -85,B 0,C 180,E1 -7840.553,E2 -7840.553} C_VEL
LIN {X 0,Y 460.468,Z 649.369,A -85,B 0,C 180,E1 -7841.446,E2 -7841.446} C_VEL
LIN {X 0,Y 460.387,Z 651.028,A -85,B 0,C 180,E1 -7843.238,E2 -7843.238} C_VEL
LIN {X 0,Y 460.389,Z 651.266,A -85,B 0,C 180,E1 -7844.139,E2 -7844.139} C_VEL
LIN {X 0,Y 460.438,Z 650.471,A -85,B 0,C 180,E1 -7845.928,E2 -7845.928} C_VEL
LIN {X 0,Y 460.528,Z 649.445,A -85,B 0,C 180,E1 -7846.857,E2 -7846.857} C_VEL
LIN {X 0,Y 460.619,Z 647.973,A -85,B 0,C 180,E1 -7847.769,E2 -7847.769} C_VEL
LIN {X 0,Y 460.816,Z 645.315,A -85,B 0,C 180,E1 -7848.991,E2 -7848.991} C_VEL
LIN {X 0,Y 461.13,Z 640.701,A -85,B 0,C 180,E1 -7850.522,E2 -7850.522} C_VEL
LIN {X 0,Y 461.465,Z 635.135,A -85,B 0,C 180,E1 -7851.926,E2 -7851.926} C_VEL
LIN {X 0,Y 461.884,Z 628.213,A -85,B 0,C 180,E1 -7853.306,E2 -7853.306} C_VEL
LIN {X 0,Y 462.352,Z 620.949,A -85,B 0,C 180,E1 -7854.471,E2 -7854.471} C_VEL
LIN {X 0,Y 462.823,Z 611.97,A -85,B 0,C 180,E1 -7855.645,E2 -7855.645} C_VEL
LIN {X 0,Y 463.253,Z 602.141,A -85,B 0,C 180,E1 -7856.689,E2 -7856.689} C_VEL
LIN {X 0,Y 463.812,Z 590.793,A -85,B 0,C 180,E1 -7857.65,E2 -7857.65} C_VEL
LIN {X 0,Y 464.239,Z 578.648,A -85,B 0,C 180,E1 -7858.443,E2 -7858.443} C_VEL
LIN {X 0,Y 464.408,Z 566.911,A -85,B 0,C 180,E1 -7859.028,E2 -7859.028} C_VEL
LIN {X 0,Y 464.545,Z 554.925,A -85,B 0,C 180,E1 -7859.453,E2 -7859.453} C_VEL
LIN {X 0,Y 464.572,Z 541.227,A -85,B 0,C 180,E1 -7859.747,E2 -7859.747} C_VEL
LIN {X 0,Y 464.944,Z 478.776,A -85,B 0,C 180,E1 -7860.738,E2 -7860.738} C_VEL
LIN {X 0,Y 460.721,Z 468.125,A -85,B 0,C 180,E1 -7861.124,E2 -7861.124} C_VEL
LIN {X 0,Y 460.536,Z 467.233,A -85,B 0,C 180,E1 -7861.287,E2 -7861.287} C_VEL
LIN {X 0,Y 460.526,Z 467.122,A -85,B 0,C 180,E1 -7864.505,E2 -7864.505} C_VEL
LIN {X 0,Y 460.505,Z 467.121,A -85,B 0,C 180,E1 -7867.624,E2 -7867.624} C_VEL
LIN {X 0,Y 460.543,Z 467.114,A -85,B 0,C 180,E1 -7870.27,E2 -7870.27} C_VEL
LIN {X 0,Y 460.501,Z 467.122,A -85,B 0,C 180,E1 -7873.377,E2 -7873.377} C_VEL
LIN {X 0,Y 460.503,Z 467.125,A -85,B 0,C 180,E1 -7876.626,E2 -7876.626} C_VEL
LIN {X 0,Y 460.547,Z 467.119,A -85,B 0,C 180,E1 -7879.732,E2 -7879.732} C_VEL
LIN {X 0,Y 460.582,Z 467.288,A -85,B 0,C 180,E1 -7881.225,E2 -7881.225} C_VEL
LIN {X 0,Y 463.191,Z 480.428,A -85,B 0,C 180,E1 -7883.532,E2 -7883.532} C_VEL
LIN {X 0,Y 462.68,Z 499.026,A -85,B 0,C 180,E1 -7886.559,E2 -7886.559} C_VEL
LIN {X 0,Y 462.106,Z 519.351,A -85,B 0,C 180,E1 -7889.828,E2 -7889.828} C_VEL
LIN {X 0,Y 464.484,Z 534.372,A -85,B 0,C 180,E1 -7890.202,E2 -7890.202} C_VEL
LIN {X 0,Y 463.419,Z 629.226,A -85,B 0,C 180,E1 -7891.809,E2 -7891.809} C_VEL
LIN {X 0,Y 463.15,Z 641.691,A -85,B 0,C 180,E1 -7892.186,E2 -7892.186} C_VEL
LIN {X 0,Y 462.705,Z 654.752,A -85,B 0,C 180,E1 -7892.77,E2 -7892.77} C_VEL
LIN {X 0,Y 462.315,Z 667.213,A -85,B 0,C 180,E1 -7893.525,E2 -7893.525} C_VEL
LIN {X 0,Y 461.834,Z 678.56,A -85,B 0,C 180,E1 -7894.419,E2 -7894.419} C_VEL
LIN {X 0,Y 461.32,Z 689.287,A -85,B 0,C 180,E1 -7895.472,E2 -7895.472} C_VEL
LIN {X 0,Y 460.874,Z 698.808,A -85,B 0,C 180,E1 -7896.642,E2 -7896.642} C_VEL
LIN {X 0,Y 460.499,Z 706.568,A -85,B 0,C 180,E1 -7897.807,E2 -7897.807} C_VEL
LIN {X 0,Y 460.183,Z 713.331,A -85,B 0,C 180,E1 -7899.049,E2 -7899.049} C_VEL
LIN {X 0,Y 459.968,Z 719.087,A -85,B 0,C 180,E1 -7900.358,E2 -7900.358} C_VEL
LIN {X 0,Y 459.786,Z 723.957,A -85,B 0,C 180,E1 -7901.785,E2 -7901.785} C_VEL
LIN {X 0,Y 459.65,Z 727.339,A -85,B 0,C 180,E1 -7903.112,E2 -7903.112} C_VEL
LIN {X 0,Y 459.577,Z 729.734,A -85,B 0,C 180,E1 -7904.458,E2 -7904.458} C_VEL
LIN {X 0,Y 459.5,Z 731.166,A -85,B 0,C 180,E1 -7905.835,E2 -7905.835} C_VEL
LIN {X 0,Y 459.515,Z 731.548,A -85,B 0,C 180,E1 -7906.738,E2 -7906.738} C_VEL
LIN {X 0,Y 459.609,Z 731.297,A -85,B 0,C 180,E1 -7908.141,E2 -7908.141} C_VEL
LIN {X 0,Y 459.621,Z 730.152,A -85,B 0,C 180,E1 -7909.427,E2 -7909.427} C_VEL
LIN {X 0,Y 459.624,Z 728.851,A -85,B 0,C 180,E1 -7910.317,E2 -7910.317} C_VEL
LIN {X 0,Y 459.792,Z 726.043,A -85,B 0,C 180,E1 -7911.651,E2 -7911.651} C_VEL
LIN {X 0,Y 459.926,Z 722.196,A -85,B 0,C 180,E1 -7912.979,E2 -7912.979} C_VEL
LIN {X 0,Y 460.089,Z 717.199,A -85,B 0,C 180,E1 -7914.302,E2 -7914.302} C_VEL
LIN {X 0,Y 460.351,Z 710.879,A -85,B 0,C 180,E1 -7915.623,E2 -7915.623} C_VEL
LIN {X 0,Y 460.686,Z 703.035,A -85,B 0,C 180,E1 -7916.94,E2 -7916.94} C_VEL
LIN {X 0,Y 461.137,Z 695.015,A -85,B 0,C 180,E1 -7918.035,E2 -7918.035} C_VEL
LIN {X 0,Y 461.614,Z 685.214,A -85,B 0,C 180,E1 -7919.128,E2 -7919.128} C_VEL
LIN {X 0,Y 462.11,Z 674.241,A -85,B 0,C 180,E1 -7920.109,E2 -7920.109} C_VEL
LIN {X 0,Y 462.56,Z 663.579,A -85,B 0,C 180,E1 -7920.871,E2 -7920.871} C_VEL
LIN {X 0,Y 462.993,Z 651.8,A -85,B 0,C 180,E1 -7921.523,E2 -7921.523} C_VEL
LIN {X 0,Y 463.326,Z 638.32,A -85,B 0,C 180,E1 -7922.065,E2 -7922.065} C_VEL
LIN {X 0,Y 463.513,Z 625.927,A -85,B 0,C 180,E1 -7922.39,E2 -7922.39} C_VEL
LIN {X 0,Y 464.63,Z 532.911,A -85,B 0,C 180,E1 -7923.998,E2 -7923.998} C_VEL
LIN {X 0,Y 462.479,Z 520.949,A -85,B 0,C 180,E1 -7924.331,E2 -7924.331} C_VEL
LIN {X 0,Y 462.591,Z 512.363,A -85,B 0,C 180,E1 -7925.668,E2 -7925.668} C_VEL
LIN {X 0,Y 463.069,Z 494.463,A -85,B 0,C 180,E1 -7928.51,E2 -7928.51} C_VEL
LIN {X 0,Y 463.302,Z 480.426,A -85,B 0,C 180,E1 -7930.71,E2 -7930.71} C_VEL
LIN {X 0,Y 461.475,Z 470.805,A -85,B 0,C 180,E1 -7932.311,E2 -7932.311} C_VEL
LIN {X 0,Y 460.582,Z 467.217,A -85,B 0,C 180,E1 -7932.973,E2 -7932.973} C_VEL
LIN {X 0,Y 460.609,Z 467.11,A -85,B 0,C 180,E1 -7935.998,E2 -7935.998} C_VEL
LIN {X 0,Y 460.575,Z 467.114,A -85,B 0,C 180,E1 -7939.616,E2 -7939.616} C_VEL
LIN {X 0,Y 460.518,Z 467.121,A -85,B 0,C 180,E1 -7942.429,E2 -7942.429} C_VEL
LIN {X 0,Y 460.554,Z 467.115,A -85,B 0,C 180,E1 -7945.796,E2 -7945.796} C_VEL
LIN {X 0,Y 460.558,Z 467.115,A -85,B 0,C 180,E1 -7948.233,E2 -7948.233} C_VEL
LIN {X 0,Y 460.529,Z 467.118,A -85,B 0,C 180,E1 -7951.282,E2 -7951.282} C_VEL
LIN {X 0,Y 460.54,Z 467.118,A -85,B 0,C 180,E1 -7954.505,E2 -7954.505} C_VEL
LIN {X 0,Y 460.509,Z 467.119,A -85,B 0,C 180,E1 -7957.623,E2 -7957.623} C_VEL
LIN {X 0,Y 460.547,Z 467.117,A -85,B 0,C 180,E1 -7960.268,E2 -7960.268} C_VEL
LIN {X 0,Y 460.507,Z 467.12,A -85,B 0,C 180,E1 -7963.375,E2 -7963.375} C_VEL
LIN {X 0,Y 460.507,Z 467.123,A -85,B 0,C 180,E1 -7966.624,E2 -7966.624} C_VEL
LIN {X 0,Y 460.546,Z 467.117,A -85,B 0,C 180,E1 -7969.73,E2 -7969.73} C_VEL
LIN {X 0,Y 460.504,Z 467.111,A -85,B 0,C 180,E1 -7972.524,E2 -7972.524} C_VEL
LIN {X 0,Y 460.542,Z 467.107,A -85,B 0,C 180,E1 -7975.622,E2 -7975.622} C_VEL
LIN {X 0,Y 460.569,Z 467.207,A -85,B 0,C 180,E1 -7979.16,E2 -7979.16} C_VEL
LIN {X 0,Y 461.504,Z 470.944,A -85,B 0,C 180,E1 -7979.83,E2 -7979.83} C_VEL
LIN {X 0,Y 464.521,Z 484.859,A -85,B 0,C 180,E1 -7982.028,E2 -7982.028} C_VEL
LIN {X 0,Y 464.646,Z 488.298,A -85,B 0,C 180,E1 -7982.526,E2 -7982.526} C_VEL
LIN {X 0,Y 463.386,Z 512.171,A -85,B 0,C 180,E1 -7985.825,E2 -7985.825} C_VEL
LIN {X 0,Y 462.472,Z 532.688,A -85,B 0,C 180,E1 -7988.608,E2 -7988.608} C_VEL
LIN {X 0,Y 461.675,Z 554.906,A -85,B 0,C 180,E1 -7991.585,E2 -7991.585} C_VEL
LIN {X 0,Y 461.406,Z 563.104,A -85,B 0,C 180,E1 -7992.631,E2 -7992.631} C_VEL
LIN {X 0,Y 464.275,Z 589.465,A -85,B 0,C 180,E1 -7993.18,E2 -7993.18} C_VEL
LIN {X 0,Y 463.546,Z 674.38,A -85,B 0,C 180,E1 -7994.528,E2 -7994.528} C_VEL
LIN {X 0,Y 463.067,Z 688.194,A -85,B 0,C 180,E1 -7994.934,E2 -7994.934} C_VEL
LIN {X 0,Y 462.566,Z 700.651,A -85,B 0,C 180,E1 -7995.48,E2 -7995.48} C_VEL
LIN {X 0,Y 461.936,Z 713.424,A -85,B 0,C 180,E1 -7996.246,E2 -7996.246} C_VEL
LIN {X 0,Y 461.361,Z 725.045,A -85,B 0,C 180,E1 -7997.143,E2 -7997.143} C_VEL
LIN {X 0,Y 460.833,Z 736.694,A -85,B 0,C 180,E1 -7998.229,E2 -7998.229} C_VEL
LIN {X 0,Y 460.545,Z 745.668,A -85,B 0,C 180,E1 -7999.225,E2 -7999.225} C_VEL
LIN {X 0,Y 460.246,Z 753.903,A -85,B 0,C 180,E1 -8000.329,E2 -8000.329} C_VEL
LIN {X 0,Y 460.017,Z 761.93,A -85,B 0,C 180,E1 -8001.653,E2 -8001.653} C_VEL
LIN {X 0,Y 459.849,Z 768.327,A -85,B 0,C 180,E1 -8002.976,E2 -8002.976} C_VEL
LIN {X 0,Y 459.801,Z 773.387,A -85,B 0,C 180,E1 -8004.297,E2 -8004.297} C_VEL
LIN {X 0,Y 459.723,Z 777.251,A -85,B 0,C 180,E1 -8005.615,E2 -8005.615} C_VEL
LIN {X 0,Y 459.778,Z 779.243,A -85,B 0,C 180,E1 -8006.493,E2 -8006.493} C_VEL
LIN {X 0,Y 459.732,Z 780.759,A -85,B 0,C 180,E1 -8007.37,E2 -8007.37} C_VEL
LIN {X 0,Y 459.724,Z 781.83,A -85,B 0,C 180,E1 -8008.246,E2 -8008.246} C_VEL
LIN {X 0,Y 459.67,Z 782.488,A -85,B 0,C 180,E1 -8009.123,E2 -8009.123} C_VEL
LIN {X 0,Y 459.706,Z 782.737,A -85,B 0,C 180,E1 -8009.999,E2 -8009.999} C_VEL
LIN {X 0,Y 459.668,Z 782.521,A -85,B 0,C 180,E1 -8010.875,E2 -8010.875} C_VEL
LIN {X 0,Y 459.719,Z 781.901,A -85,B 0,C 180,E1 -8011.751,E2 -8011.751} C_VEL
LIN {X 0,Y 459.727,Z 780.871,A -85,B 0,C 180,E1 -8012.627,E2 -8012.627} C_VEL
LIN {X 0,Y 459.767,Z 779.384,A -85,B 0,C 180,E1 -8013.504,E2 -8013.504} C_VEL
LIN {X 0,Y 459.72,Z 776.299,A -85,B 0,C 180,E1 -8014.822,E2 -8014.822} C_VEL
LIN {X 0,Y 459.771,Z 772.106,A -85,B 0,C 180,E1 -8016.141,E2 -8016.141} C_VEL
LIN {X 0,Y 459.891,Z 765.655,A -85,B 0,C 180,E1 -8017.683,E2 -8017.683} C_VEL
LIN {X 0,Y 460.087,Z 758.582,A -85,B 0,C 180,E1 -8019.006,E2 -8019.006} C_VEL
LIN {X 0,Y 460.403,Z 749.66,A -85,B 0,C 180,E1 -8020.331,E2 -8020.331} C_VEL
LIN {X 0,Y 460.753,Z 740.49,A -85,B 0,C 180,E1 -8021.436,E2 -8021.436} C_VEL
LIN {X 0,Y 461.267,Z 730.278,A -85,B 0,C 180,E1 -8022.434,E2 -8022.434} C_VEL
LIN {X 0,Y 461.792,Z 714.873,A -85,B 0,C 180,E1 -8023.643,E2 -8023.643} C_VEL
LIN {X 0,Y 462.435,Z 702.337,A -85,B 0,C 180,E1 -8024.409,E2 -8024.409} C_VEL
LIN {X 0,Y 462.921,Z 690.394,A -85,B 0,C 180,E1 -8024.955,E2 -8024.955} C_VEL
LIN {X 0,Y 463.398,Z 677.395,A -85,B 0,C 180,E1 -8025.361,E2 -8025.361} C_VEL
LIN {X 0,Y 463.637,Z 659.017,A -85,B 0,C 180,E1 -8025.691,E2 -8025.691} C_VEL
LIN {X 0,Y 464.041,Z 587.848,A -85,B 0,C 180,E1 -8026.799,E2 -8026.799} C_VEL
LIN {X 0,Y 461.399,Z 563.549,A -85,B 0,C 180,E1 -8027.298,E2 -8027.298} C_VEL
LIN {X 0,Y 462.24,Z 537.737,A -85,B 0,C 180,E1 -8030.7,E2 -8030.7} C_VEL
LIN {X 0,Y 463.067,Z 516.954,A -85,B 0,C 180,E1 -8033.476,E2 -8033.476} C_VEL
LIN {X 0,Y 464.1,Z 493.986,A -85,B 0,C 180,E1 -8036.583,E2 -8036.583} C_VEL
LIN {X 0,Y 464.453,Z 485.61,A -85,B 0,C 180,E1 -8037.728,E2 -8037.728} C_VEL
LIN {X 0,Y 462.042,Z 473.753,A -85,B 0,C 180,E1 -8039.502,E2 -8039.502} C_VEL
LIN {X 0,Y 460.56,Z 467.227,A -85,B 0,C 180,E1 -8040.551,E2 -8040.551} C_VEL
LIN {X 0,Y 460.514,Z 467.122,A -85,B 0,C 180,E1 -8043.324,E2 -8043.324} C_VEL
LIN {X 0,Y 460.459,Z 467.127,A -85,B 0,C 180,E1 -8046.529,E2 -8046.529} C_VEL
LIN {X 0,Y 460.502,Z 467.122,A -85,B 0,C 180,E1 -8049.863,E2 -8049.863} C_VEL
LIN {X 0,Y 460.47,Z 467.123,A -85,B 0,C 180,E1 -8052.894,E2 -8052.894} C_VEL
LIN {X 0,Y 460.497,Z 467.122,A -85,B 0,C 180,E1 -8055.83,E2 -8055.83} C_VEL
LIN {X 0,Y 460.51,Z 467.117,A -85,B 0,C 180,E1 -8058.986,E2 -8058.986} C_VEL
LIN {X 0,Y 460.488,Z 467.127,A -85,B 0,C 180,E1 -8062.375,E2 -8062.375} C_VEL
LIN {X 0,Y 460.534,Z 467.115,A -85,B 0,C 180,E1 -8065.622,E2 -8065.622} C_VEL
LIN {X 0,Y 460.526,Z 467.118,A -85,B 0,C 180,E1 -8068.743,E2 -8068.743} C_VEL
LIN {X 0,Y 460.565,Z 467.117,A -85,B 0,C 180,E1 -8072.254,E2 -8072.254} C_VEL
LIN {X 0,Y 460.512,Z 467.117,A -85,B 0,C 180,E1 -8075.666,E2 -8075.666} C_VEL
LIN {X 0,Y 460.508,Z 467.123,A -85,B 0,C 180,E1 -8078.577,E2 -8078.577} C_VEL
LIN {X 0,Y 460.576,Z 467.109,A -85,B 0,C 180,E1 -8081.31,E2 -8081.31} C_VEL
LIN {X 0,Y 460.591,Z 467.11,A -85,B 0,C 180,E1 -8084.058,E2 -8084.058} C_VEL
LIN {X 0,Y 460.596,Z 467.106,A -85,B 0,C 180,E1 -8087.665,E2 -8087.665} C_VEL
LIN {X 0,Y 460.614,Z 467.104,A -85,B 0,C 180,E1 -8091.223,E2 -8091.223} C_VEL
LIN {X 0,Y 460.684,Z 467.096,A -85,B 0,C 180,E1 -8093.869,E2 -8093.869} C_VEL
LIN {X 0,Y 460.785,Z 467.083,A -85,B 0,C 180,E1 -8097.377,E2 -8097.377} C_VEL
LIN {X 0,Y 460.837,Z 467.078,A -85,B 0,C 180,E1 -8100,E2 -8100} C_VEL
LIN {X 0,Y 460.809,Z 467.087,A -85,B 0,C 180,E1 -8102.622,E2 -8102.622} C_VEL
LIN {X 0,Y 460.687,Z 467.097,A -85,B 0,C 180,E1 -8106.13,E2 -8106.13} C_VEL
LIN {X 0,Y 460.615,Z 467.11,A -85,B 0,C 180,E1 -8108.776,E2 -8108.776} C_VEL
LIN {X 0,Y 460.598,Z 467.112,A -85,B 0,C 180,E1 -8112.445,E2 -8112.445} C_VEL
LIN {X 0,Y 460.585,Z 467.108,A -85,B 0,C 180,E1 -8115.998,E2 -8115.998} C_VEL
LIN {X 0,Y 460.557,Z 467.116,A -85,B 0,C 180,E1 -8118.902,E2 -8118.902} C_VEL
LIN {X 0,Y 460.502,Z 467.118,A -85,B 0,C 180,E1 -8121.486,E2 -8121.486} C_VEL
LIN {X 0,Y 460.528,Z 467.118,A -85,B 0,C 180,E1 -8124.333,E2 -8124.333} C_VEL
LIN {X 0,Y 460.57,Z 467.112,A -85,B 0,C 180,E1 -8127.244,E2 -8127.244} C_VEL
LIN {X 0,Y 460.498,Z 467.12,A -85,B 0,C 180,E1 -8130.241,E2 -8130.241} C_VEL
LIN {X 0,Y 460.516,Z 467.118,A -85,B 0,C 180,E1 -8133.326,E2 -8133.326} C_VEL
LIN {X 0,Y 460.466,Z 467.127,A -85,B 0,C 180,E1 -8136.53,E2 -8136.53} C_VEL
LIN {X 0,Y 460.533,Z 467.122,A -85,B 0,C 180,E1 -8138.899,E2 -8138.899} C_VEL
LIN {X 0,Y 460.512,Z 467.118,A -85,B 0,C 180,E1 -8142.182,E2 -8142.182} C_VEL
LIN {X 0,Y 460.511,Z 467.119,A -85,B 0,C 180,E1 -8145.413,E2 -8145.413} C_VEL
LIN {X 0,Y 460.535,Z 467.116,A -85,B 0,C 180,E1 -8148.397,E2 -8148.397} C_VEL
LIN {X 0,Y 460.537,Z 467.117,A -85,B 0,C 180,E1 -8151.27,E2 -8151.27} C_VEL
LIN {X 0,Y 460.503,Z 467.121,A -85,B 0,C 180,E1 -8154.556,E2 -8154.556} C_VEL
LIN {X 0,Y 460.523,Z 467.116,A -85,B 0,C 180,E1 -8157.717,E2 -8157.717} C_VEL
LIN {X 0,Y 460.532,Z 467.119,A -85,B 0,C 180,E1 -8160.771,E2 -8160.771} C_VEL
LIN {X 0,Y 460.556,Z 467.112,A -85,B 0,C 180,E1 -8163.736,E2 -8163.736} C_VEL
LIN {X 0,Y 460.539,Z 467.116,A -85,B 0,C 180,E1 -8166.625,E2 -8166.625} C_VEL
LIN {X 0,Y 460.547,Z 467.116,A -85,B 0,C 180,E1 -8169.454,E2 -8169.454} C_VEL
LIN {X 0,Y 460.554,Z 467.112,A -85,B 0,C 180,E1 -8172.232,E2 -8172.232} C_VEL
LIN {X 0,Y 460.561,Z 467.117,A -85,B 0,C 180,E1 -8174.966,E2 -8174.966} C_VEL
LIN {X 0,Y 460.608,Z 467.106,A -85,B 0,C 180,E1 -8178.561,E2 -8178.561} C_VEL
LIN {X 0,Y 460.574,Z 467.113,A -85,B 0,C 180,E1 -8179.243,E2 -8179.243} C_VEL
LIN {X 0,Y 459.921,Z 467.2,A -85,B 0,C 180,E1 -8179.973,E2 -8179.973} C_VEL
LIN {X 0,Y 457.103,Z 467.554,A -85,B 0,C 180,E1 -8181.159,E2 -8181.159} C_VEL
LIN {X 0,Y 454.724,Z 467.847,A -85,B 0,C 180,E1 -8182.116,E2 -8182.116} C_VEL
LIN {X 0,Y 453.713,Z 467.97,A -85,B 0,C 180,E1 -8182.855,E2 -8182.855} C_VEL
LIN {X 0,Y 453.636,Z 467.978,A -85,B 0,C 180,E1 -8183.106,E2 -8183.106} C_VEL
LIN {X 0,Y 453.671,Z 467.974,A -85,B 0,C 180,E1 -8184.668,E2 -8184.668} C_VEL
LIN {X 0,Y 453.645,Z 468.182,A -85,B 0,C 180,E1 -8186.949,E2 -8186.949} C_VEL
LIN {X 0,Y 453.967,Z 469.282,A -85,B 0,C 180,E1 -8187.09,E2 -8187.09} C_VEL
LIN {X 0,Y 457.492,Z 479.597,A -85,B 0,C 180,E1 -8187.389,E2 -8187.389} C_VEL
LIN {X 0,Y 457.149,Z 549.22,A -85,B 0,C 180,E1 -8188.511,E2 -8188.511} C_VEL
LIN {X 0,Y 457.048,Z 562.242,A -85,B 0,C 180,E1 -8188.897,E2 -8188.897} C_VEL
LIN {X 0,Y 456.882,Z 575.005,A -85,B 0,C 180,E1 -8189.461,E2 -8189.461} C_VEL
LIN {X 0,Y 456.586,Z 585.977,A -85,B 0,C 180,E1 -8190.112,E2 -8190.112} C_VEL
LIN {X 0,Y 456.159,Z 597.508,A -85,B 0,C 180,E1 -8190.995,E2 -8190.995} C_VEL
LIN {X 0,Y 455.646,Z 607.886,A -85,B 0,C 180,E1 -8191.99,E2 -8191.99} C_VEL
LIN {X 0,Y 455.267,Z 617.211,A -85,B 0,C 180,E1 -8193.099,E2 -8193.099} C_VEL
LIN {X 0,Y 454.847,Z 624.888,A -85,B 0,C 180,E1 -8194.21,E2 -8194.21} C_VEL
LIN {X 0,Y 454.465,Z 632.381,A -85,B 0,C 180,E1 -8195.548,E2 -8195.548} C_VEL
LIN {X 0,Y 454.085,Z 639.318,A -85,B 0,C 180,E1 -8197.114,E2 -8197.114} C_VEL
LIN {X 0,Y 453.807,Z 643.935,A -85,B 0,C 180,E1 -8198.462,E2 -8198.462} C_VEL
LIN {X 0,Y 453.604,Z 647.458,A -85,B 0,C 180,E1 -8199.814,E2 -8199.814} C_VEL
LIN {X 0,Y 453.483,Z 649.247,A -85,B 0,C 180,E1 -8200.719,E2 -8200.719} C_VEL
LIN {X 0,Y 453.402,Z 651.459,A -85,B 0,C 180,E1 -8202.437,E2 -8202.437} C_VEL
LIN {X 0,Y 453.371,Z 652.11,A -85,B 0,C 180,E1 -8203.447,E2 -8203.447} C_VEL
LIN {X 0,Y 453.355,Z 652.229,A -85,B 0,C 180,E1 -8204.363,E2 -8204.363} C_VEL
LIN {X 0,Y 453.422,Z 651.4,A -85,B 0,C 180,E1 -8206.057,E2 -8206.057} C_VEL
LIN {X 0,Y 453.532,Z 650.155,A -85,B 0,C 180,E1 -8207.125,E2 -8207.125} C_VEL
LIN {X 0,Y 453.755,Z 647.645,A -85,B 0,C 180,E1 -8208.514,E2 -8208.514} C_VEL
LIN {X 0,Y 454.006,Z 644.056,A -85,B 0,C 180,E1 -8209.912,E2 -8209.912} C_VEL
LIN {X 0,Y 454.315,Z 639.257,A -85,B 0,C 180,E1 -8211.319,E2 -8211.319} C_VEL
LIN {X 0,Y 454.758,Z 633.078,A -85,B 0,C 180,E1 -8212.73,E2 -8212.73} C_VEL
LIN {X 0,Y 455.227,Z 625.869,A -85,B 0,C 180,E1 -8214.047,E2 -8214.047} C_VEL
LIN {X 0,Y 455.772,Z 617.052,A -85,B 0,C 180,E1 -8215.336,E2 -8215.336} C_VEL
LIN {X 0,Y 456.319,Z 606.886,A -85,B 0,C 180,E1 -8216.53,E2 -8216.53} C_VEL
LIN {X 0,Y 456.81,Z 596.746,A -85,B 0,C 180,E1 -8217.488,E2 -8217.488} C_VEL
LIN {X 0,Y 457.289,Z 585.486,A -85,B 0,C 180,E1 -8218.329,E2 -8218.329} C_VEL
LIN {X 0,Y 457.623,Z 573.009,A -85,B 0,C 180,E1 -8219.047,E2 -8219.047} C_VEL
LIN {X 0,Y 457.758,Z 560.108,A -85,B 0,C 180,E1 -8219.585,E2 -8219.585} C_VEL
LIN {X 0,Y 457.859,Z 547.128,A -85,B 0,C 180,E1 -8219.926,E2 -8219.926} C_VEL
LIN {X 0,Y 458.295,Z 480.514,A -85,B 0,C 180,E1 -8221.008,E2 -8221.008} C_VEL
LIN {X 0,Y 453.702,Z 468.984,A -85,B 0,C 180,E1 -8221.437,E2 -8221.437} C_VEL
LIN {X 0,Y 453.53,Z 468.069,A -85,B 0,C 180,E1 -8221.624,E2 -8221.624} C_VEL
LIN {X 0,Y 453.48,Z 467.996,A -85,B 0,C 180,E1 -8224.991,E2 -8224.991} C_VEL
LIN {X 0,Y 453.464,Z 468,A -85,B 0,C 180,E1 -8228.313,E2 -8228.313} C_VEL
LIN {X 0,Y 453.498,Z 467.995,A -85,B 0,C 180,E1 -8230.61,E2 -8230.61} C_VEL
LIN {X 0,Y 453.458,Z 468,A -85,B 0,C 180,E1 -8233.245,E2 -8233.245} C_VEL
LIN {X 0,Y 453.468,Z 467.997,A -85,B 0,C 180,E1 -8235.78,E2 -8235.78} C_VEL
LIN {X 0,Y 453.484,Z 467.998,A -85,B 0,C 180,E1 -8238.21,E2 -8238.21} C_VEL
LIN {X 0,Y 453.553,Z 468.197,A -85,B 0,C 180,E1 -8241.008,E2 -8241.008} C_VEL
LIN {X 0,Y 456.282,Z 481.684,A -85,B 0,C 180,E1 -8243.395,E2 -8243.395} C_VEL
LIN {X 0,Y 455.771,Z 500.532,A -85,B 0,C 180,E1 -8246.487,E2 -8246.487} C_VEL
LIN {X 0,Y 455.2,Z 519.603,A -85,B 0,C 180,E1 -8249.576,E2 -8249.576} C_VEL
LIN {X 0,Y 457.697,Z 534.675,A -85,B 0,C 180,E1 -8249.955,E2 -8249.955} C_VEL
LIN {X 0,Y 456.554,Z 629.054,A -85,B 0,C 180,E1 -8251.592,E2 -8251.592} C_VEL
LIN {X 0,Y 456.256,Z 641.846,A -85,B 0,C 180,E1 -8251.978,E2 -8251.978} C_VEL
LIN {X 0,Y 455.805,Z 654.968,A -85,B 0,C 180,E1 -8252.572,E2 -8252.572} C_VEL
LIN {X 0,Y 455.408,Z 666.79,A -85,B 0,C 180,E1 -8253.291,E2 -8253.291} C_VEL
LIN {X 0,Y 454.92,Z 677.729,A -85,B 0,C 180,E1 -8254.143,E2 -8254.143} C_VEL
LIN {X 0,Y 454.387,Z 688.502,A -85,B 0,C 180,E1 -8255.195,E2 -8255.195} C_VEL
LIN {X 0,Y 453.96,Z 697.428,A -85,B 0,C 180,E1 -8256.265,E2 -8256.265} C_VEL
LIN {X 0,Y 453.567,Z 705.529,A -85,B 0,C 180,E1 -8257.45,E2 -8257.45} C_VEL
LIN {X 0,Y 453.18,Z 712.978,A -85,B 0,C 180,E1 -8258.796,E2 -8258.796} C_VEL
LIN {X 0,Y 452.933,Z 718.534,A -85,B 0,C 180,E1 -8260.04,E2 -8260.04} C_VEL
LIN {X 0,Y 452.733,Z 723.904,A -85,B 0,C 180,E1 -8261.569,E2 -8261.569} C_VEL
LIN {X 0,Y 452.604,Z 727.238,A -85,B 0,C 180,E1 -8262.841,E2 -8262.841} C_VEL
LIN {X 0,Y 452.492,Z 730.04,A -85,B 0,C 180,E1 -8264.362,E2 -8264.362} C_VEL
LIN {X 0,Y 452.436,Z 731.416,A -85,B 0,C 180,E1 -8265.609,E2 -8265.609} C_VEL
LIN {X 0,Y 452.417,Z 731.9,A -85,B 0,C 180,E1 -8266.526,E2 -8266.526} C_VEL
LIN {X 0,Y 452.535,Z 731.742,A -85,B 0,C 180,E1 -8268.077,E2 -8268.077} C_VEL
LIN {X 0,Y 452.556,Z 730.809,A -85,B 0,C 180,E1 -8269.26,E2 -8269.26} C_VEL
LIN {X 0,Y 452.534,Z 729.588,A -85,B 0,C 180,E1 -8270.164,E2 -8270.164} C_VEL
LIN {X 0,Y 452.695,Z 726.937,A -85,B 0,C 180,E1 -8271.519,E2 -8271.519} C_VEL
LIN {X 0,Y 452.857,Z 723.253,A -85,B 0,C 180,E1 -8272.868,E2 -8272.868} C_VEL
LIN {X 0,Y 453.016,Z 718.446,A -85,B 0,C 180,E1 -8274.213,E2 -8274.213} C_VEL
LIN {X 0,Y 453.298,Z 712.368,A -85,B 0,C 180,E1 -8275.554,E2 -8275.554} C_VEL
LIN {X 0,Y 453.629,Z 704.76,A -85,B 0,C 180,E1 -8276.892,E2 -8276.892} C_VEL
LIN {X 0,Y 454.192,Z 695.261,A -85,B 0,C 180,E1 -8278.227,E2 -8278.227} C_VEL
LIN {X 0,Y 454.699,Z 685.393,A -85,B 0,C 180,E1 -8279.336,E2 -8279.336} C_VEL
LIN {X 0,Y 455.223,Z 674.359,A -85,B 0,C 180,E1 -8280.332,E2 -8280.332} C_VEL
LIN {X 0,Y 455.691,Z 663.619,A -85,B 0,C 180,E1 -8281.105,E2 -8281.105} C_VEL
LIN {X 0,Y 456.136,Z 651.681,A -85,B 0,C 180,E1 -8281.766,E2 -8281.766} C_VEL
LIN {X 0,Y 456.467,Z 638.099,A -85,B 0,C 180,E1 -8282.317,E2 -8282.317} C_VEL
LIN {X 0,Y 456.709,Z 625.181,A -85,B 0,C 180,E1 -8282.646,E2 -8282.646} C_VEL
LIN {X 0,Y 457.872,Z 533.606,A -85,B 0,C 180,E1 -8284.278,E2 -8284.278} C_VEL
LIN {X 0,Y 455.615,Z 521.11,A -85,B 0,C 180,E1 -8284.645,E2 -8284.645} C_VEL
LIN {X 0,Y 456.281,Z 496.22,A -85,B 0,C 180,E1 -8288.638,E2 -8288.638} C_VEL
LIN {X 0,Y 456.466,Z 481.947,A -85,B 0,C 180,E1 -8290.872,E2 -8290.872} C_VEL
LIN {X 0,Y 454.589,Z 472.344,A -85,B 0,C 180,E1 -8292.5,E2 -8292.5} C_VEL
LIN {X 0,Y 453.526,Z 468.085,A -85,B 0,C 180,E1 -8293.291,E2 -8293.291} C_VEL
LIN {X 0,Y 453.553,Z 467.989,A -85,B 0,C 180,E1 -8296.196,E2 -8296.196} C_VEL
LIN {X 0,Y 453.525,Z 467.995,A -85,B 0,C 180,E1 -8299.039,E2 -8299.039} C_VEL
LIN {X 0,Y 453.485,Z 467.996,A -85,B 0,C 180,E1 -8301.836,E2 -8301.836} C_VEL
LIN {X 0,Y 453.501,Z 467.997,A -85,B 0,C 180,E1 -8304.736,E2 -8304.736} C_VEL
LIN {X 0,Y 453.538,Z 467.989,A -85,B 0,C 180,E1 -8307.959,E2 -8307.959} C_VEL
LIN {X 0,Y 453.474,Z 467.996,A -85,B 0,C 180,E1 -8311.525,E2 -8311.525} C_VEL
LIN {X 0,Y 453.496,Z 467.999,A -85,B 0,C 180,E1 -8314.777,E2 -8314.777} C_VEL
LIN {X 0,Y 453.471,Z 467.998,A -85,B 0,C 180,E1 -8318.311,E2 -8318.311} C_VEL
LIN {X 0,Y 453.502,Z 467.996,A -85,B 0,C 180,E1 -8320.608,E2 -8320.608} C_VEL
LIN {X 0,Y 453.463,Z 467.998,A -85,B 0,C 180,E1 -8323.243,E2 -8323.243} C_VEL
LIN {X 0,Y 453.472,Z 467.998,A -85,B 0,C 180,E1 -8325.778,E2 -8325.778} C_VEL
LIN {X 0,Y 453.487,Z 467.998,A -85,B 0,C 180,E1 -8328.209,E2 -8328.209} C_VEL
LIN {X 0,Y 453.478,Z 467.986,A -85,B 0,C 180,E1 -8330.796,E2 -8330.796} C_VEL
LIN {X 0,Y 453.458,Z 468.002,A -85,B 0,C 180,E1 -8333.916,E2 -8333.916} C_VEL
LIN {X 0,Y 453.482,Z 467.999,A -85,B 0,C 180,E1 -8337.15,E2 -8337.15} C_VEL
LIN {X 0,Y 453.532,Z 468.224,A -85,B 0,C 180,E1 -8338.906,E2 -8338.906} C_VEL
LIN {X 0,Y 456.462,Z 480.466,A -85,B 0,C 180,E1 -8340.947,E2 -8340.947} C_VEL
LIN {X 0,Y 457.828,Z 487.673,A -85,B 0,C 180,E1 -8342.081,E2 -8342.081} C_VEL
LIN {X 0,Y 456.677,Z 509.93,A -85,B 0,C 180,E1 -8345.228,E2 -8345.228} C_VEL
LIN {X 0,Y 455.592,Z 531.916,A -85,B 0,C 180,E1 -8348.269,E2 -8348.269} C_VEL
LIN {X 0,Y 454.641,Z 555.767,A -85,B 0,C 180,E1 -8351.523,E2 -8351.523} C_VEL
LIN {X 0,Y 454.411,Z 561.682,A -85,B 0,C 180,E1 -8352.31,E2 -8352.31} C_VEL
LIN {X 0,Y 455.629,Z 572.326,A -85,B 0,C 180,E1 -8352.566,E2 -8352.566} C_VEL
LIN {X 0,Y 457.487,Z 590.502,A -85,B 0,C 180,E1 -8352.936,E2 -8352.936} C_VEL
LIN {X 0,Y 456.727,Z 672.865,A -85,B 0,C 180,E1 -8354.262,E2 -8354.262} C_VEL
LIN {X 0,Y 456.3,Z 686.053,A -85,B 0,C 180,E1 -8354.648,E2 -8354.648} C_VEL
LIN {X 0,Y 455.773,Z 697.663,A -85,B 0,C 180,E1 -8355.145,E2 -8355.145} C_VEL
LIN {X 0,Y 455.184,Z 709.338,A -85,B 0,C 180,E1 -8355.81,E2 -8355.81} C_VEL
LIN {X 0,Y 454.612,Z 720.035,A -85,B 0,C 180,E1 -8356.59,E2 -8356.59} C_VEL
LIN {X 0,Y 454.047,Z 734.04,A -85,B 0,C 180,E1 -8357.824,E2 -8357.824} C_VEL
LIN {X 0,Y 453.632,Z 741.439,A -85,B 0,C 180,E1 -8358.606,E2 -8358.606} C_VEL
LIN {X 0,Y 453.297,Z 750.364,A -85,B 0,C 180,E1 -8359.728,E2 -8359.728} C_VEL
LIN {X 0,Y 452.999,Z 758.978,A -85,B 0,C 180,E1 -8361.073,E2 -8361.073} C_VEL
LIN {X 0,Y 452.791,Z 765.897,A -85,B 0,C 180,E1 -8362.417,E2 -8362.417} C_VEL
LIN {X 0,Y 452.69,Z 771.411,A -85,B 0,C 180,E1 -8363.76,E2 -8363.76} C_VEL
LIN {X 0,Y 452.664,Z 775.682,A -85,B 0,C 180,E1 -8365.1,E2 -8365.1} C_VEL
LIN {X 0,Y 452.688,Z 778.835,A -85,B 0,C 180,E1 -8366.438,E2 -8366.438} C_VEL
LIN {X 0,Y 452.651,Z 780.356,A -85,B 0,C 180,E1 -8367.329,E2 -8367.329} C_VEL
LIN {X 0,Y 452.657,Z 781.432,A -85,B 0,C 180,E1 -8368.219,E2 -8368.219} C_VEL
LIN {X 0,Y 452.599,Z 782.094,A -85,B 0,C 180,E1 -8369.109,E2 -8369.109} C_VEL
LIN {X 0,Y 452.629,Z 782.342,A -85,B 0,C 180,E1 -8369.999,E2 -8369.999} C_VEL
LIN {X 0,Y 452.597,Z 782.125,A -85,B 0,C 180,E1 -8370.888,E2 -8370.888} C_VEL
LIN {X 0,Y 452.653,Z 781.503,A -85,B 0,C 180,E1 -8371.778,E2 -8371.778} C_VEL
LIN {X 0,Y 452.646,Z 780.468,A -85,B 0,C 180,E1 -8372.668,E2 -8372.668} C_VEL
LIN {X 0,Y 452.676,Z 778.97,A -85,B 0,C 180,E1 -8373.559,E2 -8373.559} C_VEL
LIN {X 0,Y 452.649,Z 775.872,A -85,B 0,C 180,E1 -8374.897,E2 -8374.897} C_VEL
LIN {X 0,Y 452.69,Z 770.753,A -85,B 0,C 180,E1 -8376.484,E2 -8376.484} C_VEL
LIN {X 0,Y 452.862,Z 764.117,A -85,B 0,C 180,E1 -8378.027,E2 -8378.027} C_VEL
LIN {X 0,Y 453.089,Z 756.704,A -85,B 0,C 180,E1 -8379.372,E2 -8379.372} C_VEL
LIN {X 0,Y 453.443,Z 747.459,A -85,B 0,C 180,E1 -8380.717,E2 -8380.717} C_VEL
LIN {X 0,Y 453.849,Z 736.72,A -85,B 0,C 180,E1 -8381.952,E2 -8381.952} C_VEL
LIN {X 0,Y 454.307,Z 726.641,A -85,B 0,C 180,E1 -8382.886,E2 -8382.886} C_VEL
LIN {X 0,Y 455.037,Z 710.468,A -85,B 0,C 180,E1 -8384.077,E2 -8384.077} C_VEL
LIN {X 0,Y 455.696,Z 697.79,A -85,B 0,C 180,E1 -8384.798,E2 -8384.798} C_VEL
LIN {X 0,Y 456.204,Z 685.191,A -85,B 0,C 180,E1 -8385.324,E2 -8385.324} C_VEL
LIN {X 0,Y 456.585,Z 672.229,A -85,B 0,C 180,E1 -8385.682,E2 -8385.682} C_VEL
LIN {X 0,Y 457.217,Z 588.785,A -85,B 0,C 180,E1 -8387.011,E2 -8387.011} C_VEL
LIN {X 0,Y 454.391,Z 562.744,A -85,B 0,C 180,E1 -8387.538,E2 -8387.538} C_VEL
LIN {X 0,Y 455.21,Z 538.334,A -85,B 0,C 180,E1 -8390.798,E2 -8390.798} C_VEL
LIN {X 0,Y 456.101,Z 517.608,A -85,B 0,C 180,E1 -8393.616,E2 -8393.616} C_VEL
LIN {X 0,Y 457.142,Z 495.471,A -85,B 0,C 180,E1 -8396.652,E2 -8396.652} C_VEL
LIN {X 0,Y 457.462,Z 486.235,A -85,B 0,C 180,E1 -8397.94,E2 -8397.94} C_VEL
LIN {X 0,Y 453.538,Z 468.241,A -85,B 0,C 180,E1 -8400.727,E2 -8400.727} C_VEL
LIN {X 0,Y 453.458,Z 468.003,A -85,B 0,C 180,E1 -8401.798,E2 -8401.798} C_VEL
LIN {X 0,Y 453.468,Z 467.998,A -85,B 0,C 180,E1 -8404.988,E2 -8404.988} C_VEL
LIN {X 0,Y 453.439,Z 468.004,A -85,B 0,C 180,E1 -8408.312,E2 -8408.312} C_VEL
LIN {X 0,Y 453.462,Z 467.998,A -85,B 0,C 180,E1 -8410.61,E2 -8410.61} C_VEL
LIN {X 0,Y 453.45,Z 468.005,A -85,B 0,C 180,E1 -8414.22,E2 -8414.22} C_VEL
LIN {X 0,Y 453.439,Z 467.998,A -85,B 0,C 180,E1 -8417.002,E2 -8417.002} C_VEL
LIN {X 0,Y 453.461,Z 467.995,A -85,B 0,C 180,E1 -8419.411,E2 -8419.411} C_VEL
LIN {X 0,Y 453.439,Z 468,A -85,B 0,C 180,E1 -8422.809,E2 -8422.809} C_VEL
LIN {X 0,Y 453.465,Z 468,A -85,B 0,C 180,E1 -8426.086,E2 -8426.086} C_VEL
LIN {X 0,Y 453.464,Z 467.995,A -85,B 0,C 180,E1 -8429.239,E2 -8429.239} C_VEL
LIN {X 0,Y 453.52,Z 467.996,A -85,B 0,C 180,E1 -8432.296,E2 -8432.296} C_VEL
LIN {X 0,Y 453.483,Z 467.992,A -85,B 0,C 180,E1 -8435.263,E2 -8435.263} C_VEL
LIN {X 0,Y 453.467,Z 468.002,A -85,B 0,C 180,E1 -8438.414,E2 -8438.414} C_VEL
LIN {X 0,Y 453.509,Z 467.99,A -85,B 0,C 180,E1 -8441.008,E2 -8441.008} C_VEL
LIN {X 0,Y 453.555,Z 467.985,A -85,B 0,C 180,E1 -8443.879,E2 -8443.879} C_VEL
LIN {X 0,Y 453.55,Z 467.984,A -85,B 0,C 180,E1 -8447.47,E2 -8447.47} C_VEL
LIN {X 0,Y 453.578,Z 467.982,A -85,B 0,C 180,E1 -8451.086,E2 -8451.086} C_VEL
LIN {X 0,Y 453.652,Z 467.972,A -85,B 0,C 180,E1 -8453.774,E2 -8453.774} C_VEL
LIN {X 0,Y 453.73,Z 467.962,A -85,B 0,C 180,E1 -8457.336,E2 -8457.336} C_VEL
LIN {X 0,Y 453.807,Z 467.954,A -85,B 0,C 180,E1 -8460,E2 -8460} C_VEL
LIN {X 0,Y 453.75,Z 467.966,A -85,B 0,C 180,E1 -8462.663,E2 -8462.663} C_VEL
LIN {X 0,Y 453.655,Z 467.974,A -85,B 0,C 180,E1 -8466.225,E2 -8466.225} C_VEL
LIN {X 0,Y 453.579,Z 467.985,A -85,B 0,C 180,E1 -8468.913,E2 -8468.913} C_VEL
LIN {X 0,Y 453.549,Z 467.991,A -85,B 0,C 180,E1 -8472.529,E2 -8472.529} C_VEL
LIN {X 0,Y 453.53,Z 467.989,A -85,B 0,C 180,E1 -8476.196,E2 -8476.196} C_VEL
LIN {X 0,Y 453.506,Z 467.993,A -85,B 0,C 180,E1 -8479.041,E2 -8479.041} C_VEL
LIN {X 0,Y 453.462,Z 467.995,A -85,B 0,C 180,E1 -8481.836,E2 -8481.836} C_VEL
LIN {X 0,Y 453.5,Z 467.999,A -85,B 0,C 180,E1 -8484.735,E2 -8484.735} C_VEL
LIN {X 0,Y 453.524,Z 467.988,A -85,B 0,C 180,E1 -8487.962,E2 -8487.962} C_VEL
LIN {X 0,Y 453.453,Z 467.996,A -85,B 0,C 180,E1 -8491.526,E2 -8491.526} C_VEL
LIN {X 0,Y 453.476,Z 468.001,A -85,B 0,C 180,E1 -8494.779,E2 -8494.779} C_VEL
LIN {X 0,Y 453.461,Z 467.997,A -85,B 0,C 180,E1 -8498.312,E2 -8498.312} C_VEL
LIN {X 0,Y 453.482,Z 467.997,A -85,B 0,C 180,E1 -8500.61,E2 -8500.61} C_VEL
LIN {X 0,Y 453.465,Z 467.996,A -85,B 0,C 180,E1 -8504.221,E2 -8504.221} C_VEL
LIN {X 0,Y 453.482,Z 467.999,A -85,B 0,C 180,E1 -8507.01,E2 -8507.01} C_VEL
LIN {X 0,Y 453.523,Z 467.991,A -85,B 0,C 180,E1 -8510.556,E2 -8510.556} C_VEL
LIN {X 0,Y 453.447,Z 467.997,A -85,B 0,C 180,E1 -8513.919,E2 -8513.919} C_VEL
LIN {X 0,Y 453.474,Z 467.999,A -85,B 0,C 180,E1 -8517.153,E2 -8517.153} C_VEL
LIN {X 0,Y 453.467,Z 467.995,A -85,B 0,C 180,E1 -8520.27,E2 -8520.27} C_VEL
LIN {X 0,Y 453.502,Z 467.994,A -85,B 0,C 180,E1 -8523.296,E2 -8523.296} C_VEL
LIN {X 0,Y 453.497,Z 467.991,A -85,B 0,C 180,E1 -8526.24,E2 -8526.24} C_VEL
LIN {X 0,Y 453.478,Z 468.001,A -85,B 0,C 180,E1 -8529.119,E2 -8529.119} C_VEL
LIN {X 0,Y 453.507,Z 467.989,A -85,B 0,C 180,E1 -8531.946,E2 -8531.946} C_VEL
LIN {X 0,Y 453.536,Z 467.989,A -85,B 0,C 180,E1 -8534.728,E2 -8534.728} C_VEL
LIN {X 0,Y 453.556,Z 467.984,A -85,B 0,C 180,E1 -8538.38,E2 -8538.38} C_VEL
LIN {X 0,Y 453.649,Z 467.976,A -85,B 0,C 180,E1 -8541.987,E2 -8541.987} C_VEL
LIN {X 0,Y 453.636,Z 467.978,A -85,B 0,C 180,E1 -8543.106,E2 -8543.106} C_VEL
LIN {X 0,Y 452.956,Z 468.065,A -85,B 0,C 180,E1 -8543.599,E2 -8543.599} C_VEL
LIN {X 0,Y 450.071,Z 468.425,A -85,B 0,C 180,E1 -8544.37,E2 -8544.37} C_VEL
LIN {X 0,Y 447.16,Z 468.788,A -85,B 0,C 180,E1 -8545.15,E2 -8545.15} C_VEL
LIN {X 0,Y 446.462,Z 468.873,A -85,B 0,C 180,E1 -8545.655,E2 -8545.655} C_VEL
LIN {X 0,Y 446.544,Z 468.994,A -85,B 0,C 180,E1 -8546.674,E2 -8546.674} C_VEL
LIN {X 0,Y 446.753,Z 469.884,A -85,B 0,C 180,E1 -8546.831,E2 -8546.831} C_VEL
LIN {X 0,Y 450.767,Z 481.289,A -85,B 0,C 180,E1 -8547.174,E2 -8547.174} C_VEL
LIN {X 0,Y 450.291,Z 549.978,A -85,B 0,C 180,E1 -8548.297,E2 -8548.297} C_VEL
LIN {X 0,Y 450.21,Z 563.038,A -85,B 0,C 180,E1 -8548.688,E2 -8548.688} C_VEL
LIN {X 0,Y 449.992,Z 576.149,A -85,B 0,C 180,E1 -8549.274,E2 -8549.274} C_VEL
LIN {X 0,Y 449.693,Z 588.002,A -85,B 0,C 180,E1 -8550.001,E2 -8550.001} C_VEL
LIN {X 0,Y 449.233,Z 599.333,A -85,B 0,C 180,E1 -8550.898,E2 -8550.898} C_VEL
LIN {X 0,Y 448.712,Z 609.568,A -85,B 0,C 180,E1 -8551.909,E2 -8551.909} C_VEL
LIN {X 0,Y 448.349,Z 617.91,A -85,B 0,C 180,E1 -8552.922,E2 -8552.922} C_VEL
LIN {X 0,Y 447.911,Z 625.643,A -85,B 0,C 180,E1 -8554.05,E2 -8554.05} C_VEL
LIN {X 0,Y 447.515,Z 633.184,A -85,B 0,C 180,E1 -8555.408,E2 -8555.408} C_VEL
LIN {X 0,Y 447.155,Z 639.26,A -85,B 0,C 180,E1 -8556.771,E2 -8556.771} C_VEL
LIN {X 0,Y 446.853,Z 644.095,A -85,B 0,C 180,E1 -8558.139,E2 -8558.139} C_VEL
LIN {X 0,Y 446.632,Z 647.821,A -85,B 0,C 180,E1 -8559.512,E2 -8559.512} C_VEL
LIN {X 0,Y 446.437,Z 650.541,A -85,B 0,C 180,E1 -8560.891,E2 -8560.891} C_VEL
LIN {X 0,Y 446.357,Z 652.523,A -85,B 0,C 180,E1 -8562.526,E2 -8562.526} C_VEL
LIN {X 0,Y 446.344,Z 653.138,A -85,B 0,C 180,E1 -8563.663,E2 -8563.663} C_VEL
LIN {X 0,Y 446.345,Z 653.187,A -85,B 0,C 180,E1 -8564.593,E2 -8564.593} C_VEL
LIN {X 0,Y 446.447,Z 652.309,A -85,B 0,C 180,E1 -8566.207,E2 -8566.207} C_VEL
LIN {X 0,Y 446.547,Z 650.84,A -85,B 0,C 180,E1 -8567.401,E2 -8567.401} C_VEL
LIN {X 0,Y 446.783,Z 648.185,A -85,B 0,C 180,E1 -8568.814,E2 -8568.814} C_VEL
LIN {X 0,Y 447.084,Z 644.44,A -85,B 0,C 180,E1 -8570.234,E2 -8570.234} C_VEL
LIN {X 0,Y 447.451,Z 639.515,A -85,B 0,C 180,E1 -8571.651,E2 -8571.651} C_VEL
LIN {X 0,Y 447.932,Z 633.112,A -85,B 0,C 180,E1 -8573.096,E2 -8573.096} C_VEL
LIN {X 0,Y 448.428,Z 626.087,A -85,B 0,C 180,E1 -8574.361,E2 -8574.361} C_VEL
LIN {X 0,Y 448.913,Z 618.364,A -85,B 0,C 180,E1 -8575.503,E2 -8575.503} C_VEL
LIN {X 0,Y 449.509,Z 608.275,A -85,B 0,C 180,E1 -8576.713,E2 -8576.713} C_VEL
LIN {X 0,Y 450.035,Z 598.23,A -85,B 0,C 180,E1 -8577.685,E2 -8577.685} C_VEL
LIN {X 0,Y 450.554,Z 587.14,A -85,B 0,C 180,E1 -8578.537,E2 -8578.537} C_VEL
LIN {X 0,Y 450.915,Z 575.141,A -85,B 0,C 180,E1 -8579.25,E2 -8579.25} C_VEL
LIN {X 0,Y 451.076,Z 562.047,A -85,B 0,C 180,E1 -8579.824,E2 -8579.824} C_VEL
LIN {X 0,Y 451.183,Z 549.833,A -85,B 0,C 180,E1 -8580.168,E2 -8580.168} C_VEL
LIN {X 0,Y 451.581,Z 482.032,A -85,B 0,C 180,E1 -8581.297,E2 -8581.297} C_VEL
LIN {X 0,Y 446.666,Z 469.766,A -85,B 0,C 180,E1 -8581.768,E2 -8581.768} C_VEL
LIN {X 0,Y 446.483,Z 468.944,A -85,B 0,C 180,E1 -8581.953,E2 -8581.953} C_VEL
LIN {X 0,Y 446.429,Z 468.874,A -85,B 0,C 180,E1 -8585.054,E2 -8585.054} C_VEL
LIN {X 0,Y 446.417,Z 468.876,A -85,B 0,C 180,E1 -8588.08,E2 -8588.08} C_VEL
LIN {X 0,Y 446.431,Z 468.879,A -85,B 0,C 180,E1 -8590.919,E2 -8590.919} C_VEL
LIN {X 0,Y 446.403,Z 468.877,A -85,B 0,C 180,E1 -8593.847,E2 -8593.847} C_VEL
LIN {X 0,Y 446.403,Z 468.88,A -85,B 0,C 180,E1 -8596.405,E2 -8596.405} C_VEL
LIN {X 0,Y 446.432,Z 468.878,A -85,B 0,C 180,E1 -8599.083,E2 -8599.083} C_VEL
LIN {X 0,Y 446.527,Z 469.083,A -85,B 0,C 180,E1 -8600.781,E2 -8600.781} C_VEL
LIN {X 0,Y 449.339,Z 482.994,A -85,B 0,C 180,E1 -8603.261,E2 -8603.261} C_VEL
LIN {X 0,Y 448.931,Z 499.219,A -85,B 0,C 180,E1 -8605.946,E2 -8605.946} C_VEL
LIN {X 0,Y 448.267,Z 519.868,A -85,B 0,C 180,E1 -8609.314,E2 -8609.314} C_VEL
LIN {X 0,Y 450.875,Z 535.845,A -85,B 0,C 180,E1 -8609.732,E2 -8609.732} C_VEL
LIN {X 0,Y 449.629,Z 630.001,A -85,B 0,C 180,E1 -8611.401,E2 -8611.401} C_VEL
LIN {X 0,Y 449.311,Z 643.288,A -85,B 0,C 180,E1 -8611.824,E2 -8611.824} C_VEL
LIN {X 0,Y 448.879,Z 656.155,A -85,B 0,C 180,E1 -8612.429,E2 -8612.429} C_VEL
LIN {X 0,Y 448.426,Z 668.638,A -85,B 0,C 180,E1 -8613.221,E2 -8613.221} C_VEL
LIN {X 0,Y 447.844,Z 680.362,A -85,B 0,C 180,E1 -8614.185,E2 -8614.185} C_VEL
LIN {X 0,Y 447.342,Z 689.969,A -85,B 0,C 180,E1 -8615.165,E2 -8615.165} C_VEL
LIN {X 0,Y 446.882,Z 699.434,A -85,B 0,C 180,E1 -8616.358,E2 -8616.358} C_VEL
LIN {X 0,Y 446.457,Z 707.238,A -85,B 0,C 180,E1 -8617.559,E2 -8617.559} C_VEL
LIN {X 0,Y 446.078,Z 714.8,A -85,B 0,C 180,E1 -8618.997,E2 -8618.997} C_VEL
LIN {X 0,Y 445.853,Z 719.827,A -85,B 0,C 180,E1 -8620.19,E2 -8620.19} C_VEL
LIN {X 0,Y 445.649,Z 724.595,A -85,B 0,C 180,E1 -8621.615,E2 -8621.615} C_VEL
LIN {X 0,Y 445.503,Z 728.125,A -85,B 0,C 180,E1 -8623.032,E2 -8623.032} C_VEL
LIN {X 0,Y 445.413,Z 730.557,A -85,B 0,C 180,E1 -8624.441,E2 -8624.441} C_VEL
LIN {X 0,Y 445.357,Z 731.601,A -85,B 0,C 180,E1 -8625.375,E2 -8625.375} C_VEL
LIN {X 0,Y 445.347,Z 732.229,A -85,B 0,C 180,E1 -8626.308,E2 -8626.308} C_VEL
LIN {X 0,Y 445.455,Z 732.193,A -85,B 0,C 180,E1 -8628.014,E2 -8628.014} C_VEL
LIN {X 0,Y 445.475,Z 731.452,A -85,B 0,C 180,E1 -8629.087,E2 -8629.087} C_VEL
LIN {X 0,Y 445.45,Z 730.34,A -85,B 0,C 180,E1 -8630.006,E2 -8630.006} C_VEL
LIN {X 0,Y 445.532,Z 728.78,A -85,B 0,C 180,E1 -8630.924,E2 -8630.924} C_VEL
LIN {X 0,Y 445.735,Z 725.605,A -85,B 0,C 180,E1 -8632.298,E2 -8632.298} C_VEL
LIN {X 0,Y 445.905,Z 721.357,A -85,B 0,C 180,E1 -8633.666,E2 -8633.666} C_VEL
LIN {X 0,Y 446.124,Z 715.916,A -85,B 0,C 180,E1 -8635.03,E2 -8635.03} C_VEL
LIN {X 0,Y 446.449,Z 709.088,A -85,B 0,C 180,E1 -8636.39,E2 -8636.39} C_VEL
LIN {X 0,Y 446.952,Z 700.531,A -85,B 0,C 180,E1 -8637.747,E2 -8637.747} C_VEL
LIN {X 0,Y 447.442,Z 691.805,A -85,B 0,C 180,E1 -8638.875,E2 -8638.875} C_VEL
LIN {X 0,Y 447.98,Z 682.224,A -85,B 0,C 180,E1 -8639.888,E2 -8639.888} C_VEL
LIN {X 0,Y 448.523,Z 671.693,A -85,B 0,C 180,E1 -8640.786,E2 -8640.786} C_VEL
LIN {X 0,Y 448.978,Z 660.151,A -85,B 0,C 180,E1 -8641.57,E2 -8641.57} C_VEL
LIN {X 0,Y 449.436,Z 648.258,A -85,B 0,C 180,E1 -8642.185,E2 -8642.185} C_VEL
LIN {X 0,Y 449.773,Z 635.277,A -85,B 0,C 180,E1 -8642.659,E2 -8642.659} C_VEL
LIN {X 0,Y 449.987,Z 621.802,A -85,B 0,C 180,E1 -8642.966,E2 -8642.966} C_VEL
LIN {X 0,Y 451.223,Z 534.805,A -85,B 0,C 180,E1 -8644.552,E2 -8644.552} C_VEL
LIN {X 0,Y 448.826,Z 521.578,A -85,B 0,C 180,E1 -8644.958,E2 -8644.958} C_VEL
LIN {X 0,Y 449.427,Z 497.788,A -85,B 0,C 180,E1 -8648.77,E2 -8648.77} C_VEL
LIN {X 0,Y 449.78,Z 485.043,A -85,B 0,C 180,E1 -8650.808,E2 -8650.808} C_VEL
LIN {X 0,Y 448.084,Z 475.339,A -85,B 0,C 180,E1 -8652.455,E2 -8652.455} C_VEL
LIN {X 0,Y 446.484,Z 469.001,A -85,B 0,C 180,E1 -8653.601,E2 -8653.601} C_VEL
LIN {X 0,Y 446.497,Z 468.869,A -85,B 0,C 180,E1 -8656.459,E2 -8656.459} C_VEL
